      (*tL_Trigger_EventTime := UInt64Add64(ULINT_TO_ULARGE(tL_Sensor_TimeStamp), LREAL_TO_UINT64(fI_TriggerDistance/fI_ConveyorSpeed * 1E9));*)
        tL_Trigger_EventTime := (tL_Sensor_TimeStamp + LREAL_TO_ULINT(fI_TriggerDistance / fI_ConveyorSpeed * 1E9));
        iL_StartPos          := iI_CurrentPos;
      END_IF;

      cO_Activate     := cL_INACTIVE;
    END_IF;

    bO_Trigger        := TRUE;
    bO_Active         := TRUE;
  	bL_InhibitTrigger := TRUE;

  cL_WAITALMOSTSTART: (*Only active when bI_UsePositionTrigger=TRUE: wait until Start position almost reached, then set timestamp*)
    (*Remaining distance in [m], converted to REAL to avoid integer wrap problems*)
    fL_RemDist             := fI_TriggerDistance + (DINT_TO_REAL(iL_StartPos) - DINT_TO_REAL(iI_CurrentPos))*0.0254 / INT_TO_REAL(iI_Resolution);
    fL_PreTriggerPosition  := fC_PreTrigFactor * fL_DeltaTimeStamp * fI_ConveyorSpeed;

    IF fL_RemDist < fL_PreTriggerPosition THEN
      cL_State             := cL_WAITSTART;
    (*tL_Trigger_EventTime := UInt64Add64(ULINT_TO_ULARGE(tL_Sensor_TimeStamp), LREAL_TO_UINT64(fL_RemDist/fI_ConveyorSpeed * 1E9));*)
      tL_Trigger_EventTime := (tL_Sensor_TimeStamp + LREAL_TO_ULINT(fL_RemDist / fI_ConveyorSpeed * 1E9));
      cO_Activate          := cL_ACTIVE;  (*Arm EL2252*)
    ELSE
      cL_State     := cL_WAITALMOSTSTART;
      cO_Activate  := cL_INACTIVE;
    END_IF;
    bO_Trigger     := TRUE;
    bO_Active      := TRUE;

  cL_WAITSTART:       (*Wait until start time reached*)
  (*IF (UInt64Cmp64(tL_Trigger_EventTime, ULINT_TO_ULARGE(tL_CurrentTime)) = -1) THEN (* StartTime elapsed *)*)
    IF (tL_Trigger_EventTime < tL_CurrentTime) THEN (* StartTime elapsed *)
      cL_State     := cL_TRIGACTIVE;
      cO_Activate  := cL_INACTIVE; (*Disarm EL2252, trigger generated*)
    ELSE
      cL_State     := cL_WAITSTART;
      cO_Activate  := cL_ACTIVE;   (*Arm EL2252*)
    END_IF;

    bO_Trigger     := TRUE;
    bO_Active      := TRUE;

  cL_TRIGACTIVE:   (*Trigger high*)
    cL_State       := cL_WAITSTOP;

  (*tL_Trigger_EventTime := UInt64Add64(tL_Trigger_EventTime,LREAL_TO_UINT64(fL_TriggerLength*1E9));*)
    tL_Trigger_EventTime := (tL_Trigger_EventTime + LREAL_TO_ULINT(fL_TriggerLength * 1E9));

    cO_Activate    := cL_INACTIVE;
    bO_Trigger     := FALSE;
    bO_Active      := TRUE;

  cL_WAITSTOP:  (*Wait until trigger time has elapsed*)
  (*IF (UInt64Cmp64(tL_Trigger_EventTime, ULINT_TO_ULARGE(tL_CurrentTime)) = -1) THEN (* StopTime elapsed *)*)
    IF (tL_Trigger_EventTime < tL_CurrentTime) THEN (* StopTime elapsed *)
      cL_State     := cL_IDLE;
      cO_Activate  := cL_INACTIVE; (*Disarm EL2252, trigger generated*)
    ELSE
      cL_State     := cL_WAITSTOP;
      cO_Activate  := cL_ACTIVE;   (*Arm EL2252*)
    END_IF;

    bO_Trigger     := FALSE;
    bO_Active      := TRUE;

  ELSE  (*Default*)
    cL_State       := cL_IDLE;
    bO_Trigger     := FALSE;
    bO_Active      := FALSE;
    cO_Activate    := cL_INACTIVE;
END_CASE;

tO_Trigger_StartTime := tL_Trigger_EventTime;

(*Release inhibit trigger*)
bL_ReleaseInhibitTrigger := (iI_CurrentPos >= (iL_StartPos + iL_SubstrateLength));
fb_FTrig_ManualTeach(CLK := bI_ManualTeachTrigger);

IF ( bL_ReleaseInhibitTrigger OR fb_FTrig_ManualTeach.Q)
   AND bL_InhibitTrigger
THEN
	bL_InhibitTrigger := FALSE;
END_IF;

(********************************* END OF FB *****************************************************)

END_FUNCTION_BLOCK

// ---- POUs/Print/DefGrid/FB_ContainerDefGrid.TcPOU
FUNCTION_BLOCK FB_ContainerDefGrid EXTENDS FB_ContainerBase
VAR_INPUT
END_VAR
VAR_OUTPUT
END_VAR
VAR
  fBImageDeformation : FB_ImageDeformation;
END_VAR

fBImageDeformation();                       // call run cyclic image deformation

METHOD AbortDeformation : BOOL
VAR_INPUT
  sReason   : STRING;
  Src       : REFERENCE TO T_ErrSrc;
  bHideLog  : BOOL;
END_VAR
IF NOT bHideLog THEN
  LogWarning(F_Concat4('Abort deformation: ', sReason, ' Src: ', Src.aDescr));  // log reason
END_IF
setError(ErrDef:=EC_DefGrid.ecDefGrid_DefGridAbort, Src:=Src); // tag ct as error
fBImageDeformation.abort();  // abort deformation
StopScript(iCT:=THIS^);
END_METHOD

METHOD AddCamPoint : BOOL
VAR_INPUT
  sPoint : ST_DeformationPointAccurate;
END_VAR
AddCamPoint := fBImageDeformation.addCamPoint(sNewPoint:=sPoint);
END_METHOD

PROPERTY bLimited : BOOL
GET
bLimited := fBImageDeformation.bDeformationGridLimited;
END_GET
SET
fBImageDeformation.bDeformationGridLimited := bLimited;
END_SET
END_PROPERTY

(*
  Create a container, build very basics.
*)
METHOD Create : BOOL
VAR_INPUT
	nCTId	            : DINT;     (* a container identifier *)
	nCTIndex	        : UDINT;	  (* memory index (array index if CT in CT array) *)
END_VAR
SUPER^.Create(nCTId:=nCTId, nCTIndex:=nCTIndex);
fBImageDeformation.reset();
fBImageDeformation.nProcessId := THIS^.pCT^.iId;
END_METHOD

PROPERTY eCamMode : E_CameraMode
GET
eCamMode := fBImageDeformation.eCamMode;
END_GET
END_PROPERTY

(*
  Shift in x [SubPx]
*)
PROPERTY fDxShift : LREAL
GET
VAR
  errCtr : UDINT;
END_VAR
fDxShift := fBImageDeformation._nDxShift;
END_GET
END_PROPERTY

(*
  Shift in y [Px]
*)
PROPERTY fDyShift : LREAL
GET
VAR
  errCtr : UDINT;
END_VAR
fDyShift := fBImageDeformation._nDyShift;
END_GET
END_PROPERTY

PROPERTY fPrintLengthEffective : LREAL
GET
fPrintLengthEffective := fBImageDeformation.fPrintLengthEffective;
END_GET
SET
fBImageDeformation.fPrintLengthEffective := fPrintLengthEffective;
END_SET
END_PROPERTY

(*
  get a deformation point.
  :returns: TRUE if successful
*)
METHOD getDeformationPoint : BOOL;
VAR_INPUT
  nCol : UDINT;   // col select
  nRow : UDINT;   // row select
  nSel : UDINT;   // table selection
END_VAR
VAR_OUTPUT
  sPoint : ST_DeformationPointAccurate;
  bWasSet : BOOL;           // point was set by deformation
END_VAR
getDeformationPoint := fBImageDeformation.getDeformationPoint(nCol:=nCol, nRow:=nRow, nSel:=nSel, sPoint=>sPoint, bWasSet=>bWasSet);
END_METHOD

(*
  Deformation state of CT.
  :return:  TRUE in case of error -> any deformation error
*)
METHOD getDeformationStatus : BOOL
VAR_INPUT
END_VAR
VAR_OUTPUT
  eDStep: E_DeformationStep;// deformation step
  bDone : BOOL;             // deformation done
  bBusy : BOOL;             // deformation is busy
  nErrorId : UDINT;         // error id in case of error
  tExecutionTime : TIME;    // script update execution time?
  bAborted : BOOL;          // deformation is aborted/error
END_VAR
getDeformationStatus := fBImageDeformation.bError;

eDStep:= fBImageDeformation.eStep;
bBusy := fBImageDeformation.bBusy;
bDone := fBImageDeformation.bDone;
nErrorId := fBImageDeformation.nErrorId;
tExecutionTime := fBImageDeformation.tExecutionTime;
bAborted := fBImageDeformation.bAborted;
END_METHOD

PROPERTY LogLevel : E_LogSeverity
GET
LogLevel := SUPER^.LogLevel;
END_GET
SET
fBImageDeformation.LogLevel := LogLevel;
SUPER^.LogLevel := LogLevel;
END_SET
END_PROPERTY

PROPERTY nAvailableGridCols : UDINT
GET
nAvailableGridCols := fBImageDeformation._nGridCols;
END_GET
END_PROPERTY

PROPERTY nAvailableGridPoints : UDINT
GET
nAvailableGridPoints := fBImageDeformation.nAvailableGridPoints;
END_GET
END_PROPERTY

PROPERTY PUBLIC nRegisteredCameraPoints : UDINT
GET
nRegisteredCameraPoints := fBImageDeformation._nCamPoints;
END_GET
END_PROPERTY

PROPERTY pImageDeformation : POINTER TO FB_ImageDeformation
GET
pImageDeformation := ADR(fBImageDeformation);
END_GET
END_PROPERTY

PROPERTY sDefGridSettings : ST_DefGridSettings
GET
sDefGridSettings := fBImageDeformation.sDefGridSettings;
END_GET
END_PROPERTY

METHOD StartCamera
VAR_INPUT
  eCameraMode  : E_CameraMode;   // used camera mode
  fFeatureGrid : LREAL;          // deformation module update interval [Px]
  bResetDeformation : BOOL;      // reset current deformation state
END_VAR
// reset old deformation
IF bResetDeformation THEN
  fBImageDeformation.reset();
END_IF

// update mode
fBImageDeformation.eCamMode := eCameraMode;
fBImageDeformation.fFeatureGrid := fFeatureGrid;
fBImageDeformation.eStep := E_DeformationStep.cameraStarted;
END_METHOD

METHOD StartDeformation
VAR_INPUT
  sDefGridSettings : ST_DefGridSettings;
  fStartDeformationPos : LREAL;   // reference start position in [px]
END_VAR
fBImageDeformation.sDefGridSettings := sDefGridSettings;                  // apply grid setting
fBImageDeformation.startDeformation(                                      // start deformation process
  fStartDefPos:=fStartDeformationPos,     // reference position at current position [Px]
  fImageLength:=pJob^.fImageDepth / 1000        // fSubstrateDepth            //update with intended length
);
END_METHOD

METHOD StartScript
VAR_INPUT
  iDeformationHandler : I_DeformationHandler;
END_VAR
fBImageDeformation.iDeformationHandler := iDeformationHandler;
fBImageDeformation.eStep := E_DeformationStep.createdScriptContainer;
END_METHOD

METHOD StopScript : BOOL
VAR_INPUT
  iCT : I_CT;
END_VAR
IF fBImageDeformation.iDeformationHandler <> 0 THEN
  fBImageDeformation.iDeformationHandler.DeleteCachedCt(iCT:=iCT);
  fBImageDeformation.iDeformationHandler := 0; // remove handler after stopping (prevent further calls on same CT)
END_IF
END_METHOD

(*
  save a streamed deformation point.
  :returns: TRUE if successful
*)
METHOD storeStreamedDeformationPoint : BOOL;
VAR_INPUT
  pPoint : POINTER TO ST_DeformationPointAccurate;
END_VAR
IF pPoint = 0 THEN RETURN; END_IF

storeStreamedDeformationPoint := fBImageDeformation.storeStreamedDeformationPoint(pPoint:=pPoint);
END_METHOD

METHOD UpdateDeformation
VAR_INPUT
  fPos : LREAL; // relative deformation position in [px]
END_VAR
fBImageDeformation.updateDeformation(fPos:=fPos);
END_METHOD

END_FUNCTION_BLOCK

// ---- POUs/Print/DefGrid/FB_ImageDeformation.TcPOU
FUNCTION_BLOCK FB_ImageDeformation EXTENDS FB_PythonDeformation
VAR
  _eDeformationStep : E_DeformationStep;    // current active deformation step (handler)
  _eCameraMode      : E_CameraMode;         // active deformation mode
  _fFeatureGrid     : LREAL;                // camera feature grid [Px]
  _iDefHandler      : I_DeformationHandler; // deformation handler interface for global deformation control
  _nImgProcPoints   : DINT;                 // to calc gloabl dx/dy
  _nDxShift, _nDxSum : LREAL;               // global x grid shift
  _nDyShift, _nDySum : LREAL;               // global y grid shift
  
  // Cam points (stored locally)
  _nCamPoints        : UDINT;
  _sCamPoints        : ARRAY[0..100] OF ST_CameraPointTbl;   // received cam points
  _nCamPoint_MaxRefX : LREAL;               // max. x position of all available cam points [px]

  _sDefGridSettings  : ST_DefGridSettings;  // local copy of settings  
  // local DefGrid table [calculated]
  _sDefGridPoints    : ARRAY[0..nMAX_COLS_DEFGRID, 0..nMAX_ROWS_DEFGRID] OF ST_DeformationPointTbl; // [col, row] local grid point table
  _nGridPoints       : UDINT;               // stored and available grid points
  _nGridCols         : UDINT;               // count current complete grid columns
  // local DefGrid table [streamed]
  _sDefGridPointsStreamed : ARRAY[0..nMAX_COLS_DEFGRID, 0..nMAX_ROWS_DEFGRID] OF ST_DeformationPointTbl; // [col, row] local grid point table 
  _nGridRowsStreamed, _nGridColsStreamed : UDINT;
  
  // local grid handler(s) helper
  _nLocalGridColsGenerated: UDINT;          // already generated "local" grid columns XYR [0..x]

  _fStartDeformPos  : LREAL;                // position [Px] where deformation started on ct
  _nUpdatedGridCol  : UDINT;                // already updated grid column
  _nUpdatedFeature  : UDINT;                // number of updated features (a distance)
  _fPrintLengthOriginal  : LREAL;           // intended image depth in [m]
  _fPrintLengthEffective : LREAL;           // effective detected printing length in [m] (not yet used, but could be used for more accureate dx calculation in the future)
  _bDeformationGridLimited : BOOL;              // some deformation points were limited to a min/max boundary
  // others
  _nErrorId         : UDINT := 0;
  _sTempPoint       : ST_DeformationPointAccurate; 
END_VAR
VAR_STAT
  // sim
  eTestGridSelection : E_GridTypeSelection;
  nTestGridFactor : LREAL := 20;
END_VAR
VAR CONSTANT
  tPYTHON_TIMEOUT   : TIME  := T#500MS;     // python deformation script update response timeout  
  nMAX_COLS_DEFGRID : UDINT := 100;         // if you update this value you need to update the array variables as well (there we can't use this constant (beckhoff bug in table view))
  nMAX_ROWS_DEFGRID : UDINT := 100;         // if you update this value you need to update the array variables as well (there we can't use this constant (beckhoff bug in table view))
  nMAX_CAM_POINTS   : UDINT := 100;         // if you update this value you need to update the array variables as well (there we can't use this constant (beckhoff bug in table view))
END_VAR

IF NOT bInitialized THEN
  init();
END_IF

IF bUsePy THEN
  ExecPy();       // call python deformation handler
  
  // pull all GridPoints from FIFO and store to local table
  WHILE PopDeformationPoint(sNewPoint=>_sTempPoint) DO
    storeDeformationPoint(sPoint:=_sTempPoint);    // save point to table
  END_WHILE
END_IF

METHOD abort : BOOL
VAR_INPUT
END_VAR
_bAborted := TRUE;
END_METHOD

METHOD addCamPoint : BOOL
VAR_INPUT
  sNewPoint : ST_DeformationPointAccurate;
END_VAR
VAR
  sPointPx  : ST_DeformationPoint;
END_VAR
IF bUsePy THEN
  // push point to fifo for script
  
  addCamPoint := PushDeformationPoint(
                      sPoint:=F_EncodeDeformationPoint(sPoint:=sNewPoint, nResolution:=GVL_Deformation.nC_GridSubReso)
                 );
ELSE
  addCamPoint := TRUE;
END_IF

// store it to local table
IF addCamPoint THEN
  storeCameraPoint(sPoint:=sNewPoint); // store locally
END_IF
END_METHOD

PROPERTY bAborted : BOOL
GET
bAborted := _bAborted;
END_GET
END_PROPERTY

PROPERTY bBusy : BOOL
GET
bBusy := bPythonBusy AND NOT _bAborted;
END_GET
END_PROPERTY

PROPERTY bDeformationGridLimited : BOOL
GET
bDeformationGridLimited := _bDeformationGridLimited;
END_GET
SET
_bDeformationGridLimited := bDeformationGridLimited;
END_SET
END_PROPERTY

PROPERTY bDone : BOOL
GET
bDone := bPythonDeformationDone OR _bAborted OR (eStep = E_DeformationStep.nothing);
END_GET
END_PROPERTY

PROPERTY bError : BOOL
GET
bError := bPythonError OR _bAborted;
END_GET
END_PROPERTY

PROPERTY PRIVATE bUsePy : BOOL
GET
IF _sDefGridSettings.eDeformationType=E_DeformationType.ScriptGrid OR _sDefGridSettings.eDeformationType = E_DeformationType.ScriptGridTrend THEN
  bUsePy := TRUE;
END_IF
END_GET
END_PROPERTY

METHOD dumpGrid : BOOL
VAR_INPUT
END_VAR
END_METHOD

PROPERTY eCamMode : E_CameraMode
GET
eCamMode := _eCameraMode;
END_GET
SET
_eCameraMode := eCamMode;
END_SET
END_PROPERTY

PROPERTY eStep : E_DeformationStep
GET
eStep := _eDeformationStep;
END_GET
SET
IF eStep > _eDeformationStep THEN
  LogLvl(Lvl:=E_LogSeverity.Detail, Msg:=F_Concat4('Change deformation step: ', TO_STRING(_eDeformationStep), '->', TO_STRING(eStep)));
  _eDeformationStep := eStep;
END_IF
END_SET
END_PROPERTY

(*
  Camera feature grid. Section distance where points are detected and sent as group to PLC.
*)
PROPERTY fFeatureGrid : LREAL
GET
fFeatureGrid := _fFeatureGrid;
END_GET
SET
_fFeatureGrid := fFeatureGrid;
END_SET
END_PROPERTY

PROPERTY fPrintLengthEffective : LREAL
GET
fPrintLengthEffective := _fPrintLengthEffective;
END_GET
SET
_fPrintLengthEffective := fPrintLengthEffective;
END_SET
END_PROPERTY

// get neighbour camera point
// :returns: TRUE if present
METHOD PRIVATE getCamNeighbourPoint : BOOL
VAR_INPUT
  fPos    : LREAL;   // [px]
  nOffset : DINT;    // 0=previous, 1=next
END_VAR
VAR_OUTPUT
  Pn : ST_CameraPointTbl;
END_VAR
VAR
  i : DINT;
  foundIdx : DINT;
END_VAR
foundIdx := -1;
FOR i:=0 TO TO_DINT(_nCamPoints)-1 DO
  // previous search
  IF nOffset = 0 THEN
    IF _sCamPoints[i].sPoint.x_ref <= fpos THEN
      foundIdx := i;
    ELSE
      EXIT;
    END_IF
    
  // next searchs  
  ELSIF nOffset = 1 THEN
    IF _sCamPoints[i].sPoint.x_ref > fpos THEN
      foundIdx := i;
      EXIT;
    END_IF
  END_IF
END_FOR

IF foundIdx >= 0 THEN
  Pn := _sCamPoints[foundIdx];
  getCamNeighbourPoint := TRUE;  
END_IF
END_METHOD

// get neighbour camera point
// :returns: TRUE if present
METHOD getCamPointX : BOOL
VAR_INPUT
  nIdx : UDINT;    // 0=last, 1=first, 2=second
END_VAR
VAR_OUTPUT
  Pn : ST_CameraPointTbl;
END_VAR
IF nIdx = 0 THEN
  Pn := _sCamPoints[_nCamPoints-1];  // return first cam point
  getCamPointX := TRUE;
ELSIF nIdx <= _nCamPoints THEN
  Pn := _sCamPoints[nIdx-1];
  getCamPointX := TRUE;
ELSE
  //error
  Pn := _sCamPoints[0];   // error return first as fallback 
END_IF
END_METHOD

(*
  get a deformation point.
  :returns: TRUE if successful
*)
METHOD getDeformationPoint :  BOOL;
VAR_INPUT
  nCol : UDINT;   // col select
  nRow : UDINT;   // row select
  nSel : UDINT;   // table selection 0=GeneratedGrid, 1=StreamedGrid
END_VAR
VAR_OUTPUT
  sPoint : ST_DeformationPointAccurate;
  bWasSet : BOOL;
END_VAR
getDeformationPoint := FALSE;

IF TO_UDINT(nCol) > nMAX_COLS_DEFGRID THEN LogError(F_Concat5('getDeformationPoint: point col=', TO_STRING(nCol), ' out of table > ', TO_STRING(nMAX_COLS_DEFGRID), '')); RETURN; END_IF
IF TO_UDINT(nRow) > nMAX_ROWS_DEFGRID THEN LogError(F_Concat5('getDeformationPoint: point row=', TO_STRING(nRow), ' out of table > ', TO_STRING(nMAX_ROWS_DEFGRID), '')); RETURN; END_IF

IF nSel = 1 THEN
  sPoint  := _sDefGridPointsStreamed[nCol, nRow].sPoint;
  bWasSet := _sDefGridPointsStreamed[nCol, nRow].bSet;  
ELSE
  sPoint  := _sDefGridPoints[nCol, nRow].sPoint;
  bWasSet := _sDefGridPoints[nCol, nRow].bSet;  
END_IF

getDeformationPoint := TRUE;
END_METHOD

METHOD PROTECTED gridImgProc
VAR_INPUT
  pNewDeformationPoint	: POINTER TO ST_DeformationPointAccurate;
END_VAR
IF pNewDeformationPoint = 0 THEN RETURN; END_IF

_nDxSum := (_nDxSum + pNewDeformationPoint^.dx);
_nDySum := (_nDySum + pNewDeformationPoint^.dy);
IF _nImgProcPoints > 0 THEN
  _nDxShift := _nDxSum / _nImgProcPoints;
  _nDyShift := _nDySum / _nImgProcPoints;
END_IF
_nImgProcPoints := _nImgProcPoints + 1;
END_METHOD

PROPERTY iDeformationHandler : I_DeformationHandler
GET
iDeformationHandler := _iDefHandler;
END_GET
SET
_iDefHandler := iDeformationHandler;
END_SET
END_PROPERTY

METHOD init
VAR_INPUT
END_VAR
_fbTimeout.PT := tPYTHON_TIMEOUT;
bInitialized := TRUE;
END_METHOD

PROPERTY nAvailableCamPoints : UDINT
GET
nAvailableCamPoints := _nCamPoints;
END_GET
END_PROPERTY

PROPERTY nAvailableGridPoints : UDINT
GET
nAvailableGridPoints := _nGridPoints;
END_GET
END_PROPERTY

PROPERTY nErrorId : UDINT
GET
nErrorId := _nErrorId;
END_GET
END_PROPERTY

PROPERTY nProcessId : DINT
GET
nProcessId := nPythonId;
END_GET
SET
nPythonId := nProcessId;
END_SET
END_PROPERTY

METHOD reset
VAR_INPUT
END_VAR
SUPER^.Reset();   // reset FB_PythonDeformation

_nGridPoints := 0;
_nGridCols := 0;
_nCamPoints := 0;
_nCamPoint_MaxRefX := 0;
MEMSET(destAddr:=ADR(_sDefGridPoints), fillByte:=0, n:=SIZEOF(_sDefGridPoints));
MEMSET(destAddr:=ADR(_sCamPoints), fillByte:=0, n:=SIZEOF(_sCamPoints));
MEMSET(destAddr:=ADR(_sDefGridSettings), fillByte:=0, n:=SIZEOF(_sDefGridSettings));

MEMSET(destAddr:=ADR(_sDefGridPointsStreamed), fillByte:=0, n:=SIZEOF(_sDefGridPointsStreamed));
_nGridRowsStreamed := 0;
_nGridColsStreamed := 0;

_eDeformationStep := E_DeformationStep.nothing;
_eCameraMode := E_CameraMode.NoCorrection;
_iDefHandler := 0;
_nImgProcPoints   := 0;
_nDxShift         := 0;
_nDyShift         := 0;
_nDxSum           := 0;
_nDySum           := 0; 

_nLocalGridColsGenerated:=0;
_fStartDeformPos:=0;
_nUpdatedGridCol := 0;
_nUpdatedFeature := 0;
_nErrorId := 0;
_tExecutionTime := T#0s;
END_METHOD

PROPERTY sDefGridSettings : ST_DefGridSettings
GET
sDefGridSettings := _sDefGridSettings;
END_GET
SET
_sDefGridSettings := sDefGridSettings;
END_SET
END_PROPERTY

METHOD startDeformation
VAR_INPUT
  fStartDefPos : LREAL;  // [Px]
  fImageLength : LREAL;  // [m] original image length
END_VAR
_fStartDeformPos := fStartDefPos;
_fPrintLengthOriginal := fImageLength;
_fPrintLengthEffective := fImageLength;
_nUpdatedGridCol := 0;
_nUpdatedFeature := 0;
_nCamPoint_MaxRefX := 0;

eStep := E_DeformationStep.gridStarted;  // signal to start deformation (update process)
END_METHOD

METHOD PRIVATE storeCameraPoint
VAR_INPUT
  sPoint : ST_DeformationPointAccurate;
END_VAR
// save point with checks and log.

//-- check table overflow
IF _nCamPoints >= nMAX_CAM_POINTS THEN LogError(F_Concat3('storeCamPoint: array overflow ', TO_STRING(_nCamPoints), ' ignore point, ')); RETURN; END_IF

//-- store point
_sCamPoints[_nCamPoints].bSet := TRUE;
_sCamPoints[_nCamPoints].sPoint := sPoint;
_sCamPoints[_nCamPoints].tTime := F_GetCurDcTaskTime64();
_nCamPoints := _nCamPoints+1;

// -- max. x pos 
IF sPoint.x_ref > _nCamPoint_MaxRefX THEN
  _nCamPoint_MaxRefX := sPoint.x_ref;  // point most far in ct
END_IF
END_METHOD

METHOD PRIVATE storeDeformationPoint
VAR_INPUT
  sPoint : ST_DeformationPointAccurate;
END_VAR
// do global point img processing
gridImgProc(pNewDeformationPoint:=ADR(sPoint));

// save point with checks and log.
//-- check table overflow
IF TO_UDINT(sPoint.col) > nMAX_COLS_DEFGRID THEN LogError(F_Concat5('point col=', TO_STRING(sPoint.col), ' exceeds max=', TO_STRING(nMAX_COLS_DEFGRID), ' ignore point')); RETURN; END_IF
IF TO_UDINT(sPoint.row) > nMAX_ROWS_DEFGRID THEN LogError(F_Concat5('point row=', TO_STRING(sPoint.row), ' exceeds max=', TO_STRING(nMAX_ROWS_DEFGRID), ' ignore point')); RETURN; END_IF
  
//-- store point
_sDefGridPoints[sPoint.col, sPoint.row].bSet := TRUE;
_sDefGridPoints[sPoint.col, sPoint.row].sPoint := sPoint;
_sDefGridPoints[sPoint.col, sPoint.row].tTime := F_GetCurDcTaskTime64();
IF sPoint.x_ref = 0 THEN _sDefGridPoints[sPoint.col, sPoint.row].sPoint.x_ref := sPoint.col * TO_DINT(_sDefGridSettings.nGridPitchX); END_IF// calc x pos of grid point (if not done by script)
IF sPoint.y_ref = 0 THEN _sDefGridPoints[sPoint.col, sPoint.row].sPoint.y_ref := sPoint.row * TO_DINT(_sDefGridSettings.nGridPitchY); END_IF// calc x pos of grid point (if not done by script)
// count grid points 
_nGridPoints := _nGridPoints + 1;
// count current complete grid columns
IF _sDefGridSettings.nGridSizeY > 0 THEN
  _nGridCols := (_nGridPoints/_sDefGridSettings.nGridSizeY);
END_IF
END_METHOD

METHOD storeStreamedDeformationPoint : BOOL
VAR_INPUT
  pPoint : POINTER TO ST_DeformationPointAccurate;
END_VAR
IF pPoint = 0 THEN RETURN; END_IF
IF TO_UDINT(pPoint^.col) > nMAX_COLS_DEFGRID THEN RETURN; END_IF
IF TO_UDINT(pPoint^.row) > nMAX_ROWS_DEFGRID THEN RETURN; END_IF

_sDefGridPointsStreamed[pPoint^.col, pPoint^.row].bSet := TRUE;
_sDefGridPointsStreamed[pPoint^.col, pPoint^.row].sPoint := pPoint^;
_sDefGridPointsStreamed[pPoint^.col, pPoint^.row].tTime := F_GetCurDcTaskTime64();
IF pPoint^.x_ref = 0 THEN _sDefGridPointsStreamed[pPoint^.col, pPoint^.row].sPoint.x_ref := pPoint^.col * TO_DINT(_sDefGridSettings.nGridPitchX); END_IF// calc x pos of grid point (if not done by script)
IF pPoint^.y_ref = 0 THEN _sDefGridPointsStreamed[pPoint^.col, pPoint^.row].sPoint.y_ref := pPoint^.row * TO_DINT(_sDefGridSettings.nGridPitchY); END_IF// calc x pos of grid point (if not done by script)
_nGridColsStreamed := MAX(_nGridColsStreamed, TO_UDINT(pPoint^.col));
_nGridRowsStreamed := MAX(_nGridRowsStreamed, TO_UDINT(pPoint^.row));

storeStreamedDeformationPoint := TRUE;
END_METHOD

PROPERTY tExecutionTime : TIME
GET
tExecutionTime := _tExecutionTime;  // TODO: in case of local processor read other execution time
END_GET
END_PROPERTY

METHOD updateDeformation
VAR_INPUT
  fPos : LREAL;  // current CT position in [px]
END_VAR
VAR
  fPosRel_Deform      : LREAL;    // position relative to start deformation [px]
  fPosRel_CamFeature  : LREAL;    // theoretical feature position [feature nr](based on StartDeformation NOT real on camera)
  fPosRel_GridCol     : LREAL;    // current deformation grid number [grid nr]
  sPoint : ST_DeformationPoint;
  nCurrentCol, nCurrentFeature : UDINT;
END_VAR
// cyclic call and update deformation script
// - parameter checks
IF eStep < E_DeformationStep.gridStarted OR bDone THEN RETURN; END_IF  // nothing to do if deformation was not started
IF _sDefGridSettings.nGridSizeX = 0 THEN RETURN; END_IF
IF fFeatureGrid = 0 THEN fFeatureGrid := 1024; END_IF         // set some valid default (prevents division crash)

// - calc relative Deformation position
fPosRel_Deform     := fPos - _fStartDeformPos;
fPosRel_CamFeature := fPosRel_Deform / _fFeatureGrid;
fPosRel_GridCol    := fPosRel_Deform / _sDefGridSettings.nGridPitchX;

// - check available cam points --> current feature
//    Is this blocking when position is retracting?
IF FLOOR(fPosRel_CamFeature) > _nUpdatedFeature   // by CameraFeature pitch (to sync with reception of cam points)
   //FLOOR(fPosRel_GridCol) > _nUpdatedGridCol    // by Grid Pitch  // AND _nUpdatedGridCol <= _sDefGridSettings.nGridSizeX
THEN

  nCurrentCol := TO_UDINT(FLOOR(fPosRel_GridCol));
  nCurrentFeature :=  TO_UDINT(FLOOR(fPosRel_CamFeature));

  // debug info
  LogLvl(Lvl:=E_LogSeverity.Debug, Msg:=
    F_Concat6(
        F_Concat2('update at: ', TO_STRING(fPosRel_Deform)),
        F_Concat3(' feature(', TO_STRING(fPosRel_CamFeature), ')'),
        F_Concat2(' CamP: ', TO_STRING(_nCamPoints)),
        F_Concat2(' maxX: ', TO_STRING(_nCamPoint_MaxRefX)),
        F_Concat2(' GridP: ', TO_STRING(_nGridPoints)),
        F_Concat2(' at Col: ', TO_STRING(nCurrentCol))
    )
  );

  // - update Grid (py or local) with desired position
  IF bUsePy THEN
    IF _nCamPoints > 2 THEN
      UpdatePy(fPosition:=fPosRel_Deform);
      _nUpdatedGridCol := nCurrentCol;
      _nUpdatedFeature := nCurrentFeature;
    END_IF
  ELSIF _sDefGridSettings.eDeformationType = E_DeformationType.LocalMarks1D THEN
    updateLocal_1D_Marks(nGridCol:=nCurrentCol, nFeatureCt:=nCurrentFeature);
    _nUpdatedGridCol := nCurrentCol;
    _nUpdatedFeature := nCurrentFeature;
  END_IF
END_IF
END_METHOD

METHOD PRIVATE updateLocal_1D_Marks : BOOL
VAR_INPUT
  nGridCol : UDINT;
  nFeatureCt : UDINT;
END_VAR
VAR
  row, col : UDINT;
  ct : DINT;
  col_pos_px : LREAL;   // column position in [px]
  sTmpPoint : ST_DeformationPointAccurate;
  dx, dy : LREAL;
  generateGridForCol : BOOL;
  Pn0, Pn1 : ST_CameraPointTbl;
  pPx : POINTER TO ST_CameraPointTbl;
  bn0, bn1 : BOOL;
  bFirstCol, bLastCol : BOOL;
  fPointDist : LREAL;
  relativePosX : LREAL;
END_VAR
VAR_INST
  fTrig_Done : F_TRIG;
END_VAR
VAR CONSTANT
  fC_SignConversion : LREAL := -1; 
END_VAR
bFirstCol := SEL(nGridCol=0, FALSE, TRUE);
bLastCol  := SEL(nGridCol=_sDefGridSettings.nGridSizeX-1, FALSE, TRUE);

ct := 0;
FOR col:=_nLocalGridColsGenerated TO nGridCol DO      // loop over not yet gnerated columns 
  LogLvl(Lvl:=E_LogSeverity.Debug, Msg:= F_Concat2(F_Concat2('check grid for col: ', TO_STRING(col)), ''));
  
  col_pos_px := col * _sDefGridSettings.nGridPitchX;
  dx:=0; dy:=0;
  
  bn0 := getCamNeighbourPoint(fPos:=col_pos_px, nOffset:=0, Pn=>Pn0);
  bn1 := getCamNeighbourPoint(fPos:=col_pos_px, nOffset:=1, Pn=>Pn1);
  
  IF bn0 AND bn1 THEN
    // we have neighbour points --> interpolate displacement inbetween
    // dx/dy interpolation between previous and next cam point
    fPointDist := Pn1.sPoint.x_ref-Pn0.sPoint.x_ref;
    fPointDist := SEL(fPointDist=0, fPointDist, 1);    // avoid 0 division crash
    relativePosX := (col_pos_px-Pn0.sPoint.x_ref) / (fPointDist);    // relative position of col between two cam points
    dx := fC_SignConversion * (Pn0.sPoint.dx + (Pn1.sPoint.dx - Pn0.sPoint.dx) * relativePosX);
    dy := fC_SignConversion * (Pn0.sPoint.dy + (Pn1.sPoint.dy - Pn0.sPoint.dy) * relativePosX);
    generateGridForCol:=TRUE;
    
  ELSIF bFirstCol THEN
    // generate first col when we have a cam point -> deformation from first point
    IF    bn0 THEN dx:=fC_SignConversion*Pn0.sPoint.dx; dy:=fC_SignConversion*Pn0.sPoint.dy; generateGridForCol:=TRUE;
    ELSIF bn1 THEN dx:=fC_SignConversion*Pn1.sPoint.dx; dy:=fC_SignConversion*Pn1.sPoint.dy; generateGridForCol:=TRUE;
    END_IF
    
  ELSE
    // not framed by two points toward the end, purge colums if no valid cam point is given next
    IF nGridCol - _nLocalGridColsGenerated >= 3 OR bLastCol THEN 
      IF _nCamPoints > 1 THEN
        // calc deformation based on first and last point
        bn0 := getCamPointX(nIdx:=1, Pn=>Pn0);  // first
        bn0 := getCamPointX(nIdx:=0, Pn=>Pn1);  // last
        fPointDist := Pn1.sPoint.x_ref-Pn0.sPoint.x_ref;      // distance of the two points
        fPointDist := SEL(fPointDist=0, fPointDist, 1);                // avoid 0 division crash
        relativePosX := (col_pos_px-Pn0.sPoint.x_ref) / (fPointDist);    // relative position of col between two cam points
        dx := fC_SignConversion * (Pn0.sPoint.dx + (Pn1.sPoint.dx - Pn0.sPoint.dx) * relativePosX);
        dy := fC_SignConversion * (Pn0.sPoint.dy + (Pn1.sPoint.dy - Pn0.sPoint.dy) * relativePosX);
      ELSE
        // repeat first correction (we do not have more information)
        pPx := SEL(bn1, ADR(Pn0), ADR(Pn1));
        dx := fC_SignConversion * pPx^.sPoint.dx;
        dy := fC_SignConversion * pPx^.sPoint.dy;
      END_IF
      
      generateGridForCol := TRUE;
    END_IF    
  END_IF
  
  // SIMULATION: some test grid (overwrite calculation)
  IF eTestGridSelection <> E_GridTypeSelection.Default THEN
    CASE eTestGridSelection OF
      0: dx := dx; dy := dy;                                        // default usekeep calculated
      1: dx := dy := 0;                                             // no deformation on ct 
      2: dx := nTestGridFactor; dy := 0;                            // dx static (Factor)
      3: dx := 0; dy := nTestGridFactor;                            // dy static (Factor)
      4: dx := 0; dy := TO_LREAL(col) * nTestGridFactor;            // dx = factor * col
      5: dx := TO_LREAL(col) * nTestGridFactor; dy := 0;            // dy = factor * col
      6: dx := SEL(row=1, 0, nTestGridFactor ); dy := 0;            // dx row 1 = factor ( test BOF)
    END_CASE
    generateGridForCol := TRUE;
  END_IF  
  
  // generate grid for column  
  IF generateGridForCol THEN
    LogLvl(Lvl:=E_LogSeverity.Debug, Msg:= F_Concat6('generate grid for col: ', TO_STRING(col), ' dx=', TO_STRING(dx), '/dy=', TO_STRING(dy)));

    // check for cam points and generate grid
    FOR row:=0 TO _sDefGridSettings.nGridSizeY -1 DO    // all points per col
      //LogLvl(Lvl:=E_LogSeverity.Debug, Msg:= F_Concat2(F_Concat2('gen grid point c:', TO_STRING(col)), F_Concat2('/r:', TO_STRING(row))));
      
      // - calculate x/y shift and rotation based on available CamPoints
      sTmpPoint.index := TO_DINT(col * _sDefGridSettings.nGridSizeY + row);
      sTmpPoint.x_ref := col * _sDefGridSettings.nGridPitchX;
      sTmpPoint.y_ref := row * _sDefGridSettings.nGridPitchY;
      sTmpPoint.dx    := dx;
      sTmpPoint.dy    := dy;
      sTmpPoint.col   := TO_DINT(col);
      sTmpPoint.row   := TO_DINT(row);
      sTmpPoint.valid := TRUE;
      storeDeformationPoint(sPoint:=sTmpPoint);    // save point to table
    END_FOR
    
    _nLocalGridColsGenerated := _nLocalGridColsGenerated + 1;
  END_IF
  
END_FOR


// set state variables which would be updated in PyUpdate/PyExed
_tExecutionTime := T#2MS;
_nErrorId := 0;
bPythonError := FALSE;
bPythonBusy := SEL(_nGridPoints >= _sDefGridSettings.nGridPoints, TRUE, FALSE); // all points generated
//bPythonBusy := SEL(_nGridCols   >= _sDefGridSettings.nGridSizeX,  TRUE, FALSE);  // all columns generated

fTrig_Done(CLK:=bPythonBusy);
IF fTrig_Done.Q THEN
  ;
END_IF

bPythonDeformationDone := NOT bPythonBusy;
END_METHOD

END_FUNCTION_BLOCK

// ---- POUs/Print/DefGrid/FB_PythonDeformation.TcPOU
FUNCTION_BLOCK FB_PythonDeformation EXTENDS FB_BasePrint
VAR
  // The variables below are accessed by the Python script. Do not change their names!
  // ------------------------------------------
  //FIFO Buffers
  fbFifoCamPoints : FB_DeformationPointFIFO; // Input FIFO, do not use Pop()
	fbFifoGridPoints : FB_DeformationPointFIFO; // Output FIFO, do not use Push()

	//Handshake variables
	fPythonPosition : LREAL := 0.0; (* Current position to process - should be kept constant while Python script is executing *)
	nPythonId : DINT := 0;   (* ct id for unique trace of ct in script *)
  
	bPythonStartUpdate : BOOL := FALSE; (* Tell the script to start its execution *)
	bPythonAbort : BOOL := FALSE; (* Abort any pending operation - NOT IMPLEMENTED *)
  
	bPythonBusy : BOOL := FALSE;
	bPythonUpdateDone : BOOL := FALSE; (* Set by the script when it's done or if error occurs *)
	bPythonError : BOOL := FALSE; (* Set by the script if any error occures during execution, cleared with abort - NOT IMPLEMENTED*)
  nPythonStatus : UDINT := 0; (*Set by the script status of deformation - NOT IMPLEMENTED*)
	bPythonDeformationDone : BOOL := FALSE; (* Set by the script when deformation if finished *)
  // ------------------------------------------
  
  // internal control
  _fbTimeout : TON; (* Counter with timeout *)
	_tExecutionTime : TIME := T#0S;   (*exection time local for scoping*)
  _bAborted : BOOL;
  
END_VAR

METHOD ExecPy : BOOL
VAR_OUTPUT
  bBusy : BOOL;
  nErrId : UDINT;
END_VAR
VAR
  _sTempPoint : ST_DeformationPoint;
END_VAR
// update FIFOs (external ADS access)
fbFifoCamPoints();
fbFifoGridPoints();

// work with script
IF bPythonBusy THEN // Pending job
	IF _fbTimeout.Q THEN // Timeout occurs
		_tExecutionTime := _fbTimeout.ET;
    bPythonAbort := TRUE;   // abort (pending operation) because id did not repond within timeout
		bPythonError := TRUE;   // set internal error
		nErrId := 1;
		bPythonBusy := FALSE;
    LogError(F_Concat4('Timeout during bPythonBusy, ExecTime:', TO_STRING(_tExecutionTime), ' Err:', TO_STRING(nErrId)));
	ELSIF bPythonUpdateDone THEN //Script done
		_tExecutionTime := _fbTimeout.ET;
		bPythonBusy := FALSE;
		IF bPythonError THEN
			nErrId := 2;
      LogError(F_Concat4('Error/abort requested by py, ExecTime:', TO_STRING(_tExecutionTime), ' Err:', TO_STRING(nErrId)));
		END_IF
  ELSIF _bAborted THEN      // abort if abort request set on ct
    bPythonBusy := FALSE;
    bPythonError := TRUE;   // set internal error
    nErrId := 3;
	END_IF
ELSIF bPythonAbort THEN
	bPythonStartUpdate := FALSE;
ELSE // Update/Job done  
  bPythonAbort := FALSE;
	bPythonStartUpdate := FALSE;
	bPythonUpdateDone := FALSE;
END_IF

_fbTimeout(IN := bPythonBusy);
END_METHOD

METHOD PROTECTED PopDeformationPoint :  BOOL;
VAR_OUTPUT
  sNewPoint : ST_DeformationPointAccurate;
END_VAR
VAR
  sPoint : ST_DeformationPoint;
END_VAR
IF fbFifoGridPoints.nCount > 0 THEN
  PopDeformationPoint := fbFifoGridPoints.Pop(sGridPoint=>sPoint);
  sNewPoint := F_DecodeDeformationPoint(sPoint:=sPoint, nResolution:=GVL_Deformation.nC_GridSubReso);
ELSE
  PopDeformationPoint := FALSE;
END_IF
END_METHOD

METHOD PROTECTED PushDeformationPoint : BOOL
VAR_INPUT
  sPoint : ST_DeformationPoint;
END_VAR
PushDeformationPoint:= fbFifoCamPoints.Push(sPoint);
END_METHOD

METHOD Reset
VAR_INPUT
END_VAR
fPythonPosition := 0.0;
//nPythonId := ;
bPythonStartUpdate := FALSE;
bPythonAbort := FALSE;
bPythonBusy := FALSE;
bPythonUpdateDone := FALSE;
bPythonError := FALSE;
nPythonStatus := 0;
bPythonDeformationDone := FALSE;

_fbTimeout(IN:=FALSE);
_bAborted := FALSE;

fbFifoCamPoints.Reset();
fbFifoGridPoints.Reset();
END_METHOD

METHOD UpdatePy : BOOL
VAR_INPUT
  fPosition : LREAL;
END_VAR
IF bPythonBusy THEN // Pending job
  UpdatePy:=FALSE;
  LogLvl(Lvl:=E_LogSeverity.Debug, Msg:='Python was still busy during updateDeformation');

ELSE // Job done

  IF NOT bPythonDeformationDone AND NOT bPythonAbort THEN // Sample input
    // start a update
    fPythonPosition := fPosition * GVL_Deformation.nC_GridSubReso;
    bPythonBusy := TRUE;
    bPythonError := FALSE;

    // Start script
    bPythonStartUpdate := TRUE;      
  END_IF

  UpdatePy:=TRUE;
END_IF
END_METHOD

END_FUNCTION_BLOCK

// ---- POUs/Print/DefGrid/FB_DeformationPointFIFO.TcPOU
FUNCTION_BLOCK FB_DeformationPointFIFO
VAR_OUTPUT
	nCount    : UINT;                 // Fill level
  nBufferSize : UINT := MAX_BUFFER_SIZE;
  nBufferItemSize : UINT := BUFFER_ITEM_SIZE;
END_VAR
VAR
	sBuffer 	: ARRAY[0..(MAX_BUFFER_SIZE-1)] OF ST_DeformationPoint;
	nHeadPtr  : UINT := 0;            // Point to the first non-empty idx
	nTailPtr  : UINT := 0;            // Pointer to the first free idx
  _bError    : BOOL;
END_VAR
VAR CONSTANT
	MAX_BUFFER_SIZE   : UINT := 1000;  // max. buffer size
	BUFFER_ITEM_SIZE  : UINT := SIZEOF(ST_DeformationPoint)/4; // Divide by 4 as we packed the ST_POINT with 32bits steps
END_VAR


(* now done async in method, this was dangerous...
// FIFO level
IF nTailPtr <= nHeadPtr THEN
	nCount := nHeadPtr - nTailPtr;
ELSE
	nCount := MAX_BUFFER_SIZE + nHeadPtr - nTailPtr;
END_IF
*)

PROPERTY bError : BOOL
GET
bError := _bError;
END_GET
END_PROPERTY

(*
  Get point from fifo queue. 
  :return: TRUE on success
*)
METHOD Pop : BOOL
VAR_OUTPUT
	sGridPoint : ST_DeformationPoint;
END_VAR
IF nCount = 0 THEN
  F_LogError('FB_DeformationPointFIFO is empty, cannot return an element');
  _bError := TRUE; 
  RETURN;
END_IF

sGridPoint := sBuffer[nTailPtr];
nTailPtr := (nTailPtr + 1) MOD MAX_BUFFER_SIZE;
nCount := nCount - 1;
_bError := FALSE;
Pop := TRUE;
END_METHOD

(*
  Add a new point to the fifo queue.
  :return: TRUE on success.
*)
METHOD Push : BOOL
VAR_INPUT
	sNewPoint : ST_DeformationPoint;
END_VAR
IF nCount >= MAX_BUFFER_SIZE THEN
  F_LogError('FB_DeformationPointFIFO overflow, element ignored');
  _bError := TRUE;
  RETURN;
END_IF

sBuffer[nHeadPtr] := sNewPoint;
nHeadPtr := (nHeadPtr + 1) MOD MAX_BUFFER_SIZE;
nCount := nCount + 1;
_bError := FALSE;
Push := TRUE;
END_METHOD

METHOD Reset : BOOL
VAR_INPUT
END_VAR
nTailPtr := 0;
nHeadPtr := 0;
nCount := 0;
_bError := 0;
END_METHOD

END_FUNCTION_BLOCK

// ---- POUs/Print/DefGrid/FB_CTManagerDefGrid.TcPOU
FUNCTION_BLOCK FB_CTManagerDefGrid EXTENDS FB_CTManager
VAR
  fbContainerInstances    : ARRAY[0..nC_MAX_CTS-1] OF FB_ContainerDefGrid;   // NOTE: 0 based array like base in library
  nCtr, nIndx : UDINT;
  _LogLevelCTs : E_LogSeverity := E_LogSeverity.Info;
END_VAR

// call CT manager base
SUPER^();

// call specific CT implementation
nCtr := 0;
WHILE nCtr < nListCount DO
  nIndx := ((nListTail + nCtr) MOD nC_MAX_CTS);    // calculate element index in list
  
  // cyclic call of CT body
  fbContainerInstances[nIndx]();
  
  nCtr := nCtr + 1;
END_WHILE

updateLogLevelsCTs();

(*
  Abort CTs
*)
METHOD AbortCts : BOOL
VAR_INPUT
  iCT : I_CT;     // reference CT 
  nSel : INT;     // selection: -1=all older (created before reference), 0=current only, 1=all newer (created after reference)
  Src : REFERENCE TO T_ErrSrc;
END_VAR
VAR
  iIterCt : I_CT;
  pCtSelected : POINTER TO FB_ContainerDefGrid;
END_VAR

// WARNING: This function is NOT tested!!! 
//    TODO: remove this comments when tested

IF nSel = 0 THEN
  // Abort referenced CT
  pCtSelected := GetContainerInstance(iCT:=iCT);
  IF pCtSelected <> 0 THEN
    pCtSelected^.AbortDeformation(sReason:=F_Concat2('CTM Abort CTs Sel=', TO_STRING(nSel)), Src:=Src, bHideLog:=FALSE);
  END_IF

ELSIF nSel < 0 THEN
  // Abort previous
  iIterCt := iCT;
  WHILE iIterCt.pListPrev <> 0 DO
    // get instance and abort
    pCtSelected := GetContainerInstance(iCT:=iIterCt);
    IF pCtSelected <> 0 THEN
      pCtSelected^.AbortDeformation(sReason:=F_Concat2('CTM Abort CTs Sel=', TO_STRING(nSel)), Src:=Src, bHideLog:=FALSE);
    END_IF
    // select prev
    iIterCt := iIterCt.pListPrev;
  END_WHILE

ELSIF nSel > 0 THEN  
  // Abort next
  iIterCt := iCT;
  WHILE iIterCt.pListNext <> 0 DO
    // get instance and abort
    pCtSelected := GetContainerInstance(iCT:=iIterCt);
    IF pCtSelected <> 0 THEN
      pCtSelected^.AbortDeformation(sReason:=F_Concat2('CTM Abort CTs Sel=', TO_STRING(nSel)), Src:=Src, bHideLog:=FALSE);
    END_IF
    // select next
    iIterCt := iIterCt.pListNext;
  END_WHILE
END_IF
END_METHOD

(*
  Get specific container reference (pointer) from container interface.
*)
METHOD PUBLIC GetContainerInstance : POINTER TO FB_ContainerDefGrid
VAR_INPUT
  iCT              : I_CT;          (*container at triggered event position*)
END_VAR
VAR
  nCtSel             : UDINT;
END_VAR
IF iCT = 0 THEN LogError(Msg:='GetContainerInstance invalid container'); RETURN; END_IF
nCtSel := iCT.pCT^.nMemIndex;
IF nCtSel < nC_MAX_CTS THEN
  GetContainerInstance := ADR( fbContainerInstances[nCtSel] );
END_IF
END_METHOD

METHOD Init
VAR
  nCtr      : UDINT;
END_VAR
_LogLevelCTs := E_LogSeverity.Info;

// init FB_CTManager(base) list (interface I_CT) with specific Container instances (FBs) 
FOR nCtr := 0 TO nC_MAX_CTS-1 DO
  iContainerList[nCtr] := fbContainerInstances[nCtr];
  fbContainerInstances[nCtr].LogLevel := _LogLevelCTs;
END_FOR

// call parent init
SUPER^.InitBase(aName:='CTM', aUnit:='SubPx', bAutoDelete:=TRUE);
END_METHOD

PROPERTY sCTDefGridInstancesPath : STRING
GET
// build path tho one image deformation fb
// e.g. PRG_PRINT.fbCTM.fbContainerInstances[%id%].fBImageDeformation where %id% will be resolved later in the pyhton script.
//      array in plc lower bound is index 0
sCTDefGridInstancesPath := F_CONCAT2(THIS^.InstanceName, '.fbContainerInstances[%id%].fBImageDeformation');
END_GET
END_PROPERTY

METHOD PRIVATE updateLogLevelsCTs
VAR_INST
  _LogLvl_mem  : E_LogSeverity;
END_VAR
// logLevel update from manager to all containers
IF _LogLevelCTs <> _LogLvl_mem THEN 
  nCtr := 0;
  WHILE nCtr < nC_MAX_CTS DO
    fbContainerInstances[nCtr].LogLevel := _LogLevelCTs;
    nCtr := nCtr + 1;
  END_WHILE
END_IF

_LogLvl_mem := _LogLevelCTs;
END_METHOD

END_FUNCTION_BLOCK

// ---- POUs/Print/DefGrid/FB_CTTrackerView.TcPOU
FUNCTION_BLOCK FB_CTTrackerView
VAR_INPUT
  fX_m,  fY_m     : LREAL;            // max. x/y position [m]
  nX_px, nY_px    : DINT;             // max. x/y pixel in view
  fPxToMRatio     : LREAL;            // 
  iPrintPosition  : I_PrintPosition;  // 
END_VAR

VAR
  // helper
  bInit   : BOOL;
  nCtr    : UDINT;
  nNum    : UDINT;
  
  // config
  _pCTTracker : POINTER TO FB_CTTracker;
  _fPrintResolution : LREAL;      // [dpi]
  _fSubPixelResolution : LREAL;   // sub pixel resolution
  
  // Container view list
  iCT     : I_CT;
  aCTV    : ARRAY[1..iCPr_MAX_CONTAINER] OF FB_ContainerView;
  
  // view control
  
END_VAR
VAR CONSTANT
END_VAR

IF NOT checkConfig() THEN RETURN; END_IF    // check config

// -- show CTs -----------------------
nNum := _pCTTracker^.nCount;
FOR nCtr := 1 TO nNum DO
  // get CT interface from list
  iCT := _pCTTracker^.getCT(nIdx:=nCtr);
  IF iCT <> 0 THEN
    // set position
    aCTV[nCtr].setPos(x:=iCT.GetPosRel(iTracker:=_pCTTracker^), y:=0);

    // display
    aCTV[nCtr].bHide := FALSE;
    aCTV[nCtr]( iCT:=iCT, 
                iIdx:=UDINT_TO_UINT(iCT.pCT^.nMemIndex), 
                fPxtoMRatio:=fPxToMRatio, 
                fPosToMFactor := 0.0254 / (_fPrintResolution*_fSubPixelResolution), 
                iTracker:=_pCTTracker^);
  END_IF
END_FOR

FOR nCtr := (nNum+1) TO iCPr_MAX_CONTAINER DO
  aCTV[nCtr].iCT := 0;
  aCTV[nCtr].bHide := TRUE;
END_FOR

METHOD checkConfig : BOOL
VAR_INPUT
END_VAR
VAR_INST
  _fX_m, _fY_m   : LREAL;
  _nX_px, _nY_px : DINT; 
END_VAR
VAR
  bOK : BOOL;
END_VAR
IF NOT bInit THEN RETURN; END_IF
IF iPrintPosition = 0 THEN RETURN; END_IF

_fPrintResolution := iPrintPosition.fPrintResolution;
_fSubPixelResolution := iPrintPosition.fSubPxResolution;

// changed settings
IF _fX_m <> fX_m OR
          _fY_m <> fY_m OR
          _nX_px <> nX_px OR
          _nY_px <> nY_px THEN
  // save new config
   _fX_m := fX_m;
   _fY_m := fY_m;
   _nX_px := nX_px;
   _nY_px := nY_px;
   config();
END_IF

checkConfig := TRUE;
END_METHOD

METHOD PRIVATE config
VAR_INPUT
END_VAR
// NOTE: some config values are given only here (internally)
FOR nCtr := 1 TO iCPr_MAX_CONTAINER DO
  aCTV[nCtr].init(
    nXPosMin:=0,
    nXPosMax:= F_MeterToSubPixel(fPosMeter := fX_m, fResoSubPx := _fPrintResolution * _fSubPixelResolution),
    nYPosMin:=0,
    nYPosMax:=F_MeterToSubPixel(fPosMeter := fY_m, fResoSubPx := _fPrintResolution * _fSubPixelResolution),
    bXFlip:=TRUE,
    bYFlip:=FALSE,
    nXMinPx:=0,
    nXMaxPx:=nX_px,
    nYMinPx:=0,
    nYMaxPx:=nY_px,
  );
  aCTV[nCtr].setPos(x:=0, y:=0);
END_FOR

bInit := TRUE;
END_METHOD

METHOD init : BOOL
VAR_INPUT
  pCTTracker : POINTER TO FB_CTTracker;
END_VAR
IF pCTTracker = 0 THEN RETURN; END_IF

_pCTTracker := pCTTracker;

bInit := TRUE;
END_METHOD

END_FUNCTION_BLOCK

// ---- POUs/Print/DefGrid/FB_DropSpeedComp.TcPOU
FUNCTION_BLOCK FB_DropSpeedComp
VAR_INPUT
  fMasterSpeed         : LREAL; //[m/s]
  fDropTravelDistance  : LREAL; //[m]
END_VAR
VAR_OUTPUT
  fDropPlacementError  : LREAL;
END_VAR
VAR PERSISTENT
  _bEnable             : BOOL := TRUE;
  _fDropSpeed          : LREAL := 6;         //[m/s] DropSpeed compensation, drop speed
  _fDropSpeedDeadTime  : LREAL := 0.388889;  //[ms]  DropSpeed compensation, additional dead time
END_VAR
VAR
  bCalcDeadTime        : BOOL;
  fTestSpeed           : ARRAY[1..2] OF LREAL;  // [m/min] speed at which test was done [SpeedTest1, SpeedTest2]
  fTestDisplacement    : ARRAY[1..2] OF LREAL;  // [um] measured displacement after test [MesureTest1, MeasureTest2]
  fDiffSpeed : LREAL;
  fDiffPlace : LREAL;
END_VAR

(*Speed compensation*)
IF _bEnable AND (_fDropSpeed > 0) THEN
	fDropPlacementError :=  (  (fDropTravelDistance / _fDropSpeed)
                        + (_fDropSpeedDeadTime / 1000))             (*[s]*)
                        * fMasterSpeed;
ELSE
  fDropPlacementError := 0;
END_IF;

// calculate add/dead time
IF bCalcDeadTime THEN bCalcDeadTime := FALSE;
  calcDeadTime();
END_IF

{attribute 'monitoring':='call'}
PROPERTY bEnable : BOOL
GET
bEnable := _bEnable;
END_GET
SET
_bEnable := bEnable;
END_SET
END_PROPERTY

METHOD PRIVATE calcDeadTime : BOOL
VAR_INPUT
END_VAR
fDiffSpeed :=  ( fTestSpeed[2] - fTestSpeed[1] ) * 1/60;
fDiffPlace :=  ( fTestDisplacement[2] - fTestDisplacement[1] ) * 1/1_000_000;

IF fDiffSpeed <> 0 THEN   // avoid crash
  // calc time
  _fDropSpeedDeadTime := 
  (
      fDiffPlace      // displacement diff
    * 1/fDiffSpeed    // speed diff
  ) * 1000;           // [s] -> [ms]
ELSE
  F_LogError('DropSpeedComp invalid TestSpeed given -> DeadTime not updated');
END_IF


// reset entries
fTestSpeed[2] := fTestSpeed[1] := 0;
fTestDisplacement[2] := fTestDisplacement[1] := 0;
END_METHOD

{attribute 'monitoring':='call'}
PROPERTY fDropSpeed : LREAL
GET
fDropSpeed := _fDropSpeed;
END_GET
SET
_fDropSpeed := fDropSpeed;
END_SET
END_PROPERTY

{attribute 'monitoring':='call'}
PROPERTY fDropSpeedDeadTime : LREAL
GET
fDropSpeedDeadTime := _fDropSpeedDeadTime;
END_GET
SET
_fDropSpeedDeadTime := fDropSpeedDeadTime;
END_SET
END_PROPERTY

END_FUNCTION_BLOCK

// ---- POUs/Print/DefGrid/FB_FineAlignement.TcPOU
(*
  This fb handles mechanical print unit corrections.
  - a 4p grid distortion
  - print unit bar banana correction
  NOTE: temperature extention of whole printbar is still handled in camera
*)
FUNCTION_BLOCK FB_FineAlignement EXTENDS FB_BasePrint IMPLEMENTS I_GridPointCorrection
VAR
  // config
  _fPxResolution     : LREAL; // pixel resolution

  // corrections
  //-- 4 point PU deformation correction/distortion
  //    VISU setup point providing reference and correction (NOTE: persists settings internally)
  _fbPlcCorrPoints : ARRAY[1..4] OF FB_PointCorr;
  //-- banana correction
  _fT1 : LREAL;   // temperature 1
  _fT2 : LREAL;   // temperature 2
  _dx_middle : LREAL;  // correction in middle (for view only)
  _y_max : LREAL; // print unit width [mm]
  //-- PUC 4p correction
  _pAdsCam           : POINTER TO FB_ADS_CAMERA;  // camera interface PUC
  aPucPointNames : ARRAY[1..4] OF STRING := ['1','2','3','4'];
  
  // helper
  lCtr     : UDINT;
  
  // unit test & debug
  _bUT_4p, _bUT_banana, _bUT_4pPuc : BOOL;
  _sUTPoints_dx : ARRAY[0..nC_UT_cols, 0..nC_UT_rows] OF LREAL;
  _sUTPoints_dy : ARRAY[0..nC_UT_cols, 0..nC_UT_rows] OF LREAL;
  // 4pPUC
  bSelect : ARRAY[1..4] OF BOOL;
  bSelected : ARRAY[1..4] OF BOOL;
  nSelectedPoint : UDINT;
  bXPlus, bXMinus, bYPlus, bYMinus : BOOL;
END_VAR
VAR PERSISTENT
  //-- 4point correction
  _bEnable_4p    : BOOL := FALSE;
  _bEnablePuc_4p : BOOL := FALSE;
  //  persistence of points see: FB_PointCorr
  //-- banana correction
  _bEnable_banana : BOOL := FALSE;
  _e_max_per_deltaT : LREAL := 0.01;  // [mm/°C]  TODO: use from config
END_VAR
VAR CONSTANT
  // Unit test configuration
  nC_UT_cols : DINT := 6;   // for test only
  nC_UT_rows : DINT := 5;   // for test only
END_VAR

// cyclic caluclation and view updates
//        NOTE: deformation is happening in updateCorrection() callback

//-- 4p correction
//   visu overrides (limitation rectancular point definition)
_fbPlcCorrPoints[3].fX_Ref := _fbPlcCorrPoints[1].fX_Ref;
_fbPlcCorrPoints[4].fX_Ref := _fbPlcCorrPoints[2].fX_Ref;
_fbPlcCorrPoints[2].fY_Ref := _fbPlcCorrPoints[1].fY_Ref;
_fbPlcCorrPoints[4].fY_Ref := _fbPlcCorrPoints[3].fY_Ref;
//   update CorrectionPoints view elements
FOR lCtr := 1 TO 4 DO
  _fbPlcCorrPoints[lCtr](); 
END_FOR

//-- banana correction
// just calculate the dx in the middle of the PU, just for the VISU
calc_banana_correction(x_pos:=0, y_pos:=_y_max/(2*1000), fT1:=_fT1, fT2:=_fT2, dx_corr=>_dx_middle);
_dx_middle := _dx_middle * 1000; // [m] --> [mm] for visu

// Unit test
IF _bUT_4p THEN _bUT_4p := FALSE; _test_4p(); END_IF
IF _bUT_banana THEN _bUT_banana := FALSE; _test_banana(); END_IF
IF _bUT_4pPuc THEN _test_Puc4p(); END_IF

METHOD PRIVATE _test_4p
VAR
  sPoint : ST_DeformationPoint;
  nCol, nRow, nCrPoint : DINT;
  dx, dy : LREAL;       // correction in [m]
  dx_px, dy_px : DINT;  // correction in [px]
  pPUC_CorrPointsInd : POINTER TO ARRAY[1..4] OF ST_CORRECTION_POINT;
  
  nCorrectionX : ARRAY[1..4] OF REAL := [-0.25, -0.2, 0.35, 0.35];
  nCorrectionY : ARRAY[1..4] OF REAL := [-0.45, -0.3, -0.8, -0.65];
  nCorrectionPointX_PLC : ARRAY[1..4] OF REAL := [0, 1000,   0, 1000];
  nCorrectionPointY_PLC : ARRAY[1..4] OF REAL := [0,   0, 702, 702];
  nCorrectionPointX_PUC : ARRAY[1..4] OF REAL := [0, 671.99,   0, 671.99];
  nCorrectionPointY_PUC : ARRAY[1..4] OF REAL := [-0.0001666666, -0.0001666666, 754.2108, 754.2108];
END_VAR
// setup test correcton points location for PLC & PUC 4p testing
pPUC_CorrPointsInd := _pAdsCam^.pCorrectionPointsIndication;
IF pPUC_CorrPointsInd = 0 THEN F_Report_Error(ErrType:=EN_REPORT_ERROR_TYPE.Report_Error_0Pointer);  RETURN; END_IF

FOR nCrPoint:=1 TO 4 DO
  // correction point location
  // -- PLC
  _fbPlcCorrPoints[nCrPoint].fX_Ref := nCorrectionPointX_PLC[nCrPoint];
  _fbPlcCorrPoints[nCrPoint].fY_Ref := nCorrectionPointY_PLC[nCrPoint];
  // -- PUC  
  pPUC_CorrPointsInd^[nCrPoint].posx := nCorrectionPointX_PUC[nCrPoint];
  pPUC_CorrPointsInd^[nCrPoint].posy := nCorrectionPointY_PUC[nCrPoint];
  
  // point correction  
  // -- PLC
  _fbPlcCorrPoints[nCrPoint].fX := nCorrectionX[nCrPoint];
  _fbPlcCorrPoints[nCrPoint].fY := nCorrectionY[nCrPoint];
  // -- PUC
  pPUC_CorrPointsInd^[nCrPoint].x := nCorrectionX[nCrPoint];
  pPUC_CorrPointsInd^[nCrPoint].y := nCorrectionY[nCrPoint];
END_FOR

// generate internal test grid
FOR nCol:=0 TO nC_UT_cols DO
  FOR nRow:=0 TO nC_UT_rows DO
    sPoint.col := nCol;
    sPoint.row := nRow;
    sPoint.x_ref := nCol * TO_DINT(GVL_Deformation.nC_DefaultGridPitch_X);
    sPoint.y_ref := nRow * TO_DINT(GVL_Deformation.nC_DefaultGridPitch_Y);
    sPoint.dx := 0;   // no previous deformation
    sPoint.dy := 0;   // no previous deformation
    
    // calc 4p PLC correction and apply to point
    calc_4p_correction(
        x_pos:=F_SubPixelToMeter(lPosSubPx:=sPoint.x_ref, fResSubPx:=_fPxResolution), 
        y_pos:=F_SubPixelToMeter(lPosSubPx:=sPoint.y_ref, fResSubPx:=_fPxResolution), 
        dx_corr=>dx, 
        dy_corr=>dy);
    LogInfo(
      F_Concat4(
        '4p PLC: point:', 
        F_Concat4(' x=', TO_STRING(sPoint.x_ref), '/y=', TO_STRING(sPoint.y_ref)),
        F_Concat2(' dx=', TO_STRING(dx)),
        F_Concat2(' dy=', TO_STRING(dy))
      )
    );

    // --- store in table for verification with Excel caluculation
    dx_px := F_MeterToSubPixel(fPosMeter:=dx, fResoSubPx:=_fPxResolution);
    dy_px := F_MeterToSubPixel(fPosMeter:=dy, fResoSubPx:=_fPxResolution);
    // save corrected point
    _sUTPoints_dx[nCol, nRow] := dx_px;
    _sUTPoints_dy[nCol, nRow] := dy_px;
    // print corrected point
    LogInfo(
      F_Concat4(
        F_Concat4('[c/r] ', TO_STRING(sPoint.col), '/', TO_STRING(sPoint.row)),
        F_Concat7(' dx: ', TO_STRING(sPoint.dx), '>', TO_STRING(dx_px), ' (', TO_STRING(dx), ')'),
        F_Concat7(' dy: ', TO_STRING(sPoint.dy), '>', TO_STRING(dy_px), ' (', TO_STRING(dy), ')'),
        SEL(sPoint.dx<>dx_px OR sPoint.dy<>dy_px,'',' !!!')
      )
    );
    // ---------------------------------
    
    // calc 4p PUC correction and apply to point
    calc_PUC_4p_correction(
        x_pos:=F_SubPixelToMeter(lPosSubPx:=sPoint.x_ref, fResSubPx:=_fPxResolution), 
        y_pos:=F_SubPixelToMeter(lPosSubPx:=sPoint.y_ref, fResSubPx:=_fPxResolution), 
        dx_corr=>dx, 
        dy_corr=>dy);
    LogInfo(
      F_Concat4(
        '4p PUC: point:', 
        F_Concat4(' x=', TO_STRING(sPoint.x_ref), '/y=', TO_STRING(sPoint.y_ref)),
        F_Concat2(' dx=', TO_STRING(dx)),
        F_Concat2(' dy=', TO_STRING(dy))
      )
    );

  END_FOR  
END_FOR
END_METHOD

METHOD PRIVATE _test_banana
VAR
  sPoint : ST_DeformationPoint;
  nCol, nRow : DINT;
  dx, dy : LREAL;       // correction in [m]
  dx_px, dy_px : LREAL;  // correction in [px]
END_VAR
// generate internal grid
FOR nCol:=0 TO nC_UT_cols DO
  FOR nRow:=0 TO nC_UT_rows DO
    sPoint.col := nCol;
    sPoint.row := nRow;
    sPoint.x_ref := nCol * TO_DINT(GVL_Deformation.nC_DefaultGridPitch_X);
    sPoint.y_ref := nRow * TO_DINT(GVL_Deformation.nC_DefaultGridPitch_Y);
    sPoint.dx := 0;   // no previous deformation
    sPoint.dy := 0;   // no previous deformation
    
    // calc correction and apply to point
    calc_banana_correction(
        x_pos:=F_SubPixelToMeter(lPosSubPx:=sPoint.x_ref, fResSubPx:=_fPxResolution), 
        Y_pos:=F_SubPixelToMeter(lPosSubPx:=sPoint.y_ref, fResSubPx:=_fPxResolution),
        fT1 := 68,
        fT2 := 48, 
        dx_corr=>dx
    );
    dx_px := dx;
    dy_px := dy;
    // save corrected point (dx @y-pos)
    _sUTPoints_dx[nCol, nRow] := dx_px;
    _sUTPoints_dy[nCol, nRow] := F_SubPixelToMeter(lPosSubPx:=sPoint.y_ref, fResSubPx:=_fPxResolution)*1000;
    
    // print corrected point
    LogInfo(
      F_Concat4(
        F_Concat4('[c/r] ', TO_STRING(sPoint.col), '/', TO_STRING(sPoint.row)),
        F_Concat6(' dx: ', TO_STRING(sPoint.dx), '>', TO_STRING(TO_DINT(dx_px)), ' [', TO_STRING(dx)),
        F_Concat6('  dy: ', TO_STRING(sPoint.dy), '>', TO_STRING(TO_DINT(dy_px)), ' [', TO_STRING(dy)),
        SEL(sPoint.dx<>dx_px OR sPoint.dy<>dy_px,'',' !!!')
      )
    );
  END_FOR  
END_FOR
END_METHOD

METHOD PRIVATE _test_Puc4p
VAR
  i : UDINT;

  pPUC_CorrPointsInd : POINTER TO ARRAY[1..4] OF ST_CORRECTION_POINT;
  pPoint : POINTER TO ST_CORRECTION_POINT;
END_VAR
pPUC_CorrPointsInd := _pAdsCam^.pCorrectionPointsIndication;      // get points array from ADS
IF pPUC_CorrPointsInd = 0 THEN F_Report_Error(ErrType:=EN_REPORT_ERROR_TYPE.Report_Error_0Pointer);  RETURN; END_IF

// do selection
IF    bSelect[1] THEN bSelect[1]:=FALSE; MEMSET(destAddr:=ADR(bSelected), fillByte:=0, n:=SIZEOF(bSelected)); bSelected[1] := TRUE; nSelectedPoint:=1;
ELSIF bSelect[2] THEN bSelect[2]:=FALSE; MEMSET(destAddr:=ADR(bSelected), fillByte:=0, n:=SIZEOF(bSelected)); bSelected[2] := TRUE; nSelectedPoint:=2;
ELSIF bSelect[3] THEN bSelect[3]:=FALSE; MEMSET(destAddr:=ADR(bSelected), fillByte:=0, n:=SIZEOF(bSelected)); bSelected[3] := TRUE; nSelectedPoint:=3;
ELSIF bSelect[4] THEN bSelect[4]:=FALSE; MEMSET(destAddr:=ADR(bSelected), fillByte:=0, n:=SIZEOF(bSelected)); bSelected[4] := TRUE; nSelectedPoint:=4;
END_IF

IF    bSelected[1] THEN pPoint := ADR(pPUC_CorrPointsInd^[1]);
ELSIF bSelected[2] THEN pPoint := ADR(pPUC_CorrPointsInd^[2]);
ELSIF bSelected[3] THEN pPoint := ADR(pPUC_CorrPointsInd^[3]);
ELSIF bSelected[4] THEN pPoint := ADR(pPUC_CorrPointsInd^[4]);
ELSE                    pPoint := ADR(pPUC_CorrPointsInd^[1]);
END_IF

IF bXPlus  THEN bXPlus  := FALSE; pPoint^.x := pPoint^.x + 0.05; END_IF
IF bXMinus THEN bXMinus := FALSE; pPoint^.x := pPoint^.x - 0.05; END_IF
IF bYPlus  THEN bYPlus  := FALSE; pPoint^.y := pPoint^.y + 0.05; END_IF
IF bYMinus THEN bYMinus := FALSE; pPoint^.y := pPoint^.y - 0.05; END_IF
END_METHOD

(*
  Calculate grid point displacement for a distortion with 4 rectangular defined points.
  Uses 2-bilinear interpolation between the 4 rectancular reference points.
*)
METHOD PRIVATE calc_4p_correction : BOOL
VAR_INPUT
  x_pos   : LREAL;    // point x position [m]
  y_pos   : LREAL;    // point y position [m]
END_VAR
VAR_OUTPUT
  dx_corr : LREAL;    // point correction x [m]
  dy_corr : LREAL;    // point correction y [m]
END_VAR
VAR
  dx, dy : LREAL;     // difference between Calibration Points (rectangle)
  x1, x2, y1, y2 : LREAL;
  cx1, cx2, cy1, cy2 : LREAL;
  GPx, GPy : LREAL;
  CVx, CVy : LREAL;
  lErrCtr : UDINT;
END_VAR

// Grid point position
GPx := x_pos; 
GPy := y_pos;

// Interpolation in x
x1 := _fbPlcCorrPoints[1].fX_Ref / 1000;    // [mm -> m]
x2 := _fbPlcCorrPoints[2].fX_Ref / 1000;    // [mm -> m]
dx := x2-x1;
IF dx = 0 THEN (*F_Report_Error(ErrType:=EN_REPORT_ERROR_TYPE.Report_Error_0Pointer);*) RETURN; END_IF

cx1 := (x2-GPx)/dx * (_fbPlcCorrPoints[1].fX / 1000) + (GPx-x1)/dx * (_fbPlcCorrPoints[2].fX / 1000);
cx2 := (x2-GPx)/dx * (_fbPlcCorrPoints[3].fX / 1000) + (GPx-x1)/dx * (_fbPlcCorrPoints[4].fX / 1000);
cy1 := (x2-GPx)/dx * (_fbPlcCorrPoints[1].fY / 1000) + (GPx-x1)/dx * (_fbPlcCorrPoints[2].fY / 1000);
cy2 := (x2-GPx)/dx * (_fbPlcCorrPoints[3].fY / 1000) + (GPx-x1)/dx * (_fbPlcCorrPoints[4].fY / 1000);

// Interpolation in y
y1 := _fbPlcCorrPoints[1].fY_Ref / 1000;    // [mm -> m]
y2 := _fbPlcCorrPoints[3].fY_Ref / 1000;    // [mm -> m]
dy := y2-y1;
IF dy = 0 THEN (*F_Report_Error(ErrType:=EN_REPORT_ERROR_TYPE.Report_Error_0Pointer);*) RETURN; END_IF

// Calc interpolated 
CVx := (y2 - GPy)/dy * cx1 + (GPy-y1)/dy * cx2;
CVy := (y2 - GPy)/dy * cy1 + (GPy-y1)/dy * cy2;

// return accurate new correction only
dx_corr := CVx;
dy_corr := CVy;

calc_4p_correction := TRUE;
END_METHOD

(*
  Calculate grid point displacement for print unit banana deformation.
  2nd order approximation.
*)
METHOD PRIVATE calc_banana_correction : BOOL
VAR_INPUT
  x_pos   : LREAL;    // point x position [m]
  y_pos   : LREAL;    // point y position [m]
  fT1     : LREAL;    // temperature 1 [°C]
  fT2     : LREAL;    // temperature 2 [°C]
END_VAR
VAR_OUTPUT
  dx_corr : LREAL;    // point correction x [m]
END_VAR
VAR
  delta_T : LREAL;   // delta temperature
  e_max   : LREAL;   //
  a : LREAL;
  x_dash, y_dash : LREAL;
END_VAR
IF _y_max = 0 THEN RETURN; END_IF

x_dash := y_pos * 1000; // [m] -> [mm]

delta_T := fT2-fT1;
e_max   := delta_T * _e_max_per_deltaT;

a := 4 * e_max /  EXPT(_y_max, 2);
y_dash := a * EXPT(x_dash - (_y_max / 2), 2) - e_max;

// correction value
dx_corr := (y_dash / 1000);  // [mm] -> [m]

calc_banana_correction := TRUE;
END_METHOD

(*
  Calculate grid point displacement for a distortion with 4 rectangular defined points.
  Uses 2-bilinear interpolation between the 4 rectancular reference points.
*)
METHOD PRIVATE calc_PUC_4p_correction : BOOL
VAR_INPUT
  x_pos   : LREAL;    // point x position [m]
  y_pos   : LREAL;    // point y position [m]
END_VAR
VAR_OUTPUT
  dx_corr : LREAL;    // point correction x [m]
  dy_corr : LREAL;    // point correction y [m]
END_VAR
VAR
  dx, dy : LREAL;     // difference between Calibration Points (rectangle)
  x1, x2, y1, y2 : LREAL;
  cx1, cx2, cy1, cy2 : LREAL;
  GPx, GPy : LREAL;
  CVx, CVy : LREAL;
  lErrCtr : UDINT;
  
  pPUC_CorrPointsInd : POINTER TO ARRAY[1..4] OF ST_CORRECTION_POINT;
END_VAR
VAR CONSTANT
  fTranslateX : REAL := 1;
  fTranslateY : REAL := -1;
END_VAR
pPUC_CorrPointsInd := _pAdsCam^.pCorrectionPointsIndication;      // get points array from ADS
IF pPUC_CorrPointsInd = 0 THEN F_Report_Error(ErrType:=EN_REPORT_ERROR_TYPE.Report_Error_0Pointer);  RETURN; END_IF

// NOTE: the anchor points (poyx,posy) of the PUC points are set in WorkerCamera.mJobStart!

// Grid point position
GPx := x_pos; 
GPy := y_pos;

// Interpolation in x
x1 := pPUC_CorrPointsInd^[1].posx / 1000;    // [mm -> m]
x2 := pPUC_CorrPointsInd^[2].posx / 1000;    // [mm -> m]
dx := x2-x1;
IF dx = 0 THEN (*F_Report_Error(ErrType:=EN_REPORT_ERROR_TYPE.Report_Error_0Pointer);*) RETURN; END_IF

cx1 := (x2-GPx)/dx * ((pPUC_CorrPointsInd^[1].x * fTranslateX) / 1000) + (GPx-x1)/dx * ((pPUC_CorrPointsInd^[2].x * fTranslateX) / 1000);
cx2 := (x2-GPx)/dx * ((pPUC_CorrPointsInd^[3].x * fTranslateX) / 1000) + (GPx-x1)/dx * ((pPUC_CorrPointsInd^[4].x * fTranslateX) / 1000);
cy1 := (x2-GPx)/dx * ((pPUC_CorrPointsInd^[1].y * fTranslateY) / 1000) + (GPx-x1)/dx * ((pPUC_CorrPointsInd^[2].y * fTranslateY) / 1000);
cy2 := (x2-GPx)/dx * ((pPUC_CorrPointsInd^[3].y * fTranslateY) / 1000) + (GPx-x1)/dx * ((pPUC_CorrPointsInd^[4].y * fTranslateY) / 1000);

// Interpolation in y
y1 := pPUC_CorrPointsInd^[1].posy / 1000;    // [mm -> m]
y2 := pPUC_CorrPointsInd^[3].posy / 1000;    // [mm -> m]
dy := y2-y1;
IF dy = 0 THEN (*F_Report_Error(ErrType:=EN_REPORT_ERROR_TYPE.Report_Error_0Pointer);*) RETURN; END_IF

// Calc interpolated 
CVx := (y2 - GPy)/dy * cx1 + (GPy-y1)/dy * cx2;
CVy := (y2 - GPy)/dy * cy1 + (GPy-y1)/dy * cy2;

// return accurate new correction only
dx_corr := CVx;
dy_corr := CVy;

calc_PUC_4p_correction := TRUE;
END_METHOD

PROPERTY fT_PL1 : LREAL
SET
_fT1 := fT_PL1;
END_SET
END_PROPERTY

PROPERTY fT_PL2 : LREAL
SET
_fT2 := fT_PL2;
END_SET
END_PROPERTY

METHOD init : BOOL
VAR_INPUT
  pAdsCam        : POINTER TO FB_ADS_CAMERA;  // camera interface PUC
  fPxReso        : LREAL;   // pixel resolution
  fPuWidth       : LREAL;   // Print unit width [m]
END_VAR
_fPxResolution := fPxReso;
_y_max         := fPuWidth * 1000;  // -> [mm]
_pAdsCam       := pAdsCam;
IF _pAdsCam = 0 THEN LogError('missing _pAdsCam, ads interface unknown, call worker specific init before'); END_IF

// PU Deformation
_fbPlcCorrPoints[1].init(aName:='P1', aUnit:='mm', fX_Min:=-5, fX_Max:=5, fY_Min:=-5, fY_Max:=5, fIncrStep:=0.05, 
                        bButnInvertX:=TRUE, bButnInvertY:=TRUE, bValInvertX:=TRUE, bValInvertY:=FALSE);
_fbPlcCorrPoints[2].init(aName:='P2', aUnit:='mm', fX_Min:=-5, fX_Max:=5, fY_Min:=-5, fY_Max:=5, fIncrStep:=0.05,
                        bButnInvertX:=TRUE, bButnInvertY:=TRUE, bValInvertX:=TRUE, bValInvertY:=FALSE);
_fbPlcCorrPoints[3].init(aName:='P3', aUnit:='mm', fX_Min:=-5, fX_Max:=5, fY_Min:=-5, fY_Max:=5, fIncrStep:=0.05,
                        bButnInvertX:=TRUE, bButnInvertY:=TRUE, bValInvertX:=TRUE, bValInvertY:=FALSE);
_fbPlcCorrPoints[4].init(aName:='P4', aUnit:='mm', fX_Min:=-5, fX_Max:=5, fY_Min:=-5, fY_Max:=5, fIncrStep:=0.05,
                        bButnInvertX:=TRUE, bButnInvertY:=TRUE, bValInvertX:=TRUE, bValInvertY:=FALSE);
END_METHOD

(*
  Apply fine-alignement corrections to DefGrid point
*)
METHOD updateCorrection : BOOL
VAR_INPUT
  pPoint : POINTER TO ST_DeformationPointAccurate;
END_VAR
VAR
  x_pos, dx_corr, dx_tmp : LREAL; // [m]
  y_pos, dy_corr, dy_tmp : LREAL; // [m]
END_VAR
// grid point position
x_pos := F_SubPixelToMeter(lPosSubPx:=FC_LREAL_TO_DINT(pPoint^.x_ref), fResSubPx:=_fPxResolution);  // [px -> m] 
y_pos := F_SubPixelToMeter(lPosSubPx:=FC_LREAL_TO_DINT(pPoint^.y_ref), fResSubPx:=_fPxResolution);  // [px -> m]
dx_corr := 0;
dy_corr := 0;

// calc - 4 point sheet deformation (PU and machine mechanical distortions)
IF _bEnable_4p THEN
  calc_4p_correction(x_pos:=x_pos, y_pos:=y_pos, dx_corr=>dx_tmp, dy_corr=>dy_tmp);
  dx_corr := dx_tmp + dx_corr;
  dy_corr := dy_tmp + dy_corr;
END_IF

IF _bEnablePuc_4p THEN  (*PUC 4P correction used*)
  calc_PUC_4p_correction(x_pos:=x_pos, y_pos:=y_pos, dx_corr=>dx_tmp, dy_corr=>dy_tmp);
  dx_corr := dx_tmp + dx_corr;
  dy_corr := dy_tmp + dy_corr;
END_IF

// calc - banana correction
IF _bEnable_banana THEN
  calc_banana_correction(x_pos:=x_pos, y_pos:=y_pos, fT1:=_fT1, fT2:=_fT2, dx_corr=>dx_tmp);
  dx_corr := dx_tmp + dx_corr;
END_IF
// apply new correction to deformation correction 
pPoint^.dx := pPoint^.dx + F_MeterToSubPixelReal(fPosMeter:=dx_corr, fResoSubPx:=_fPxResolution);
pPoint^.dy := pPoint^.dy + F_MeterToSubPixelReal(fPosMeter:=dy_corr, fResoSubPx:=_fPxResolution);

updateCorrection := TRUE;
END_METHOD

END_FUNCTION_BLOCK

// ---- POUs/Print/DefGrid/FB_PointCorr.TcPOU
FUNCTION_BLOCK FB_PointCorr
VAR PERSISTENT
  _fX_Pos, _fX_Ref : LREAL;   // x position (correction / reference)
  _fY_Pos, _fY_Ref : LREAL;   // y position (correction / reference)
END_VAR
VAR
  bCmd_X_minus : BOOL;    // command x minus
  bCmd_X_plus  : BOOL;    // command x plus
  bCmd_Y_minus : BOOL;    // command y minus
  bCmd_Y_plus  : BOOL;    // command y plus
  bAny         : BOOL;    // any pressed
  tSlow, tFast : TON;
  rTrig        : R_TRIG;
  nIncr        : LREAL;
  nBtnColor    : UDINT;
  // settings (init)
  _aName       : STRING(3);   // name of element
  _aUnit       : STRING(10);  // element intended [unit]
  _fX_Min, _fX_Max : LREAL;   // limit x
  _fY_Min, _fY_Max : LREAL;   // limit y
  _fIncrStep    : LREAL;      // incr. step slow (stay on button), fast *10
  _bButnInvertX, _bButnInvertY : BOOL;  // change buttons
  _bValInvertX, _bValInvertY   : BOOL;  // value *-1
END_VAR
VAR CONSTANT
  RED          : UDINT := 16#FFFF0000;
  GREEN        : UDINT := 16#FF00FF00;
END_VAR

bAny := bCmd_X_minus OR bCmd_X_plus OR bCmd_Y_minus OR bCmd_Y_plus;
rTrig(CLK:=bAny);
tSlow(IN:=bAny AND NOT tSlow.Q, PT:=T#500MS);
tFast(IN:=bAny AND NOT rTrig.Q, PT:=T#2S);

IF    tFast.Q AND tSlow.Q THEN nIncr := 10*_fIncrStep;
ELSIF tSlow.Q OR rTrig.Q THEN nIncr := _fIncrStep;
ELSE               nIncr := 0;
END_IF

nBtnColor := GREEN;
//    button pressed     increment +/-                show limit
IF    (bCmd_X_minus AND NOT _bButnInvertX) OR (bCmd_X_plus  AND _bButnInvertX) THEN _fX_Pos := _fX_Pos - nIncr; IF _fX_Pos<=_fX_Min THEN nBtnColor:=RED; END_IF
ELSIF (bCmd_X_plus  AND NOT _bButnInvertX) OR (bCmd_X_minus AND _bButnInvertX) THEN _fX_Pos := _fX_Pos + nIncr; IF _fX_Pos>=_fX_Max THEN nBtnColor:=RED; END_IF
ELSIF (bCmd_Y_minus AND NOT _bButnInvertY) OR (bCmd_Y_plus  AND _bButnInvertY) THEN _fY_Pos := _fY_Pos - nIncr; IF _fY_Pos<=_fY_Min THEN nBtnColor:=RED; END_IF
ELSIF (bCmd_Y_plus  AND NOT _bButnInvertY) OR (bCmd_Y_minus AND _bButnInvertY) THEN _fY_Pos := _fY_Pos + nIncr; IF _fY_Pos>=_fY_Max THEN nBtnColor:=RED; END_IF
END_IF

// apply limit
IF _fX_Pos<=_fX_Min THEN _fX_Pos:=_fX_Min; END_IF
IF _fX_Pos>=_fX_Max THEN _fX_Pos:=_fX_Max; END_IF
IF _fY_Pos<=_fY_Min THEN _fY_Pos:=_fY_Min; END_IF
IF _fY_Pos>=_fY_Max THEN _fY_Pos:=_fY_Max; END_IF

(*correction value in X*)
PROPERTY fX : LREAL
GET
fX := SEL(_bValInvertX, _fX_Pos, -1*_fX_Pos);
END_GET
SET
_fX_Pos := SEL(_bValInvertX, fX, -1*fX);
END_SET
END_PROPERTY

PROPERTY fX_Ref : LREAL
GET
fX_Ref := _fX_Ref;
END_GET
SET
_fX_Ref := fX_Ref;
END_SET
END_PROPERTY

(*correction value in Y*)
PROPERTY fY : LREAL
GET
fY := SEL(_bValInvertY, _fY_Pos, -1*_fY_Pos);
END_GET
SET
_fY_Pos := SEL(_bValInvertY, fY, -1*fY);
END_SET
END_PROPERTY

PROPERTY fY_Ref : LREAL
GET
fY_Ref := _fY_Ref;
END_GET
SET
_fY_Ref := fY_Ref;
END_SET
END_PROPERTY

METHOD init : BOOL
VAR_INPUT
  aName : STRING(3);       // name
  aUnit : STRING(10);      // display unit
  fX_Min, fX_Max : LREAL;  // Limits
  fY_Min, fY_Max : LREAL;  // Limits
  fIncrStep      : LREAL;  // Increment step (slow) VISU
  bButnInvertX, bButnInvertY : BOOL;  // change buttons
  bValInvertX,  bValInvertY  : BOOL;  // value *-1
END_VAR
_aName := aName;
_aUnit := aUnit;
_fX_Min := fX_Min; _fX_Max := fX_Max;
_fY_Min := fY_Min; _fY_Max := fY_Max;
_fIncrStep := fIncrStep;
_bButnInvertX := bButnInvertX;
_bButnInvertY := bButnInvertY;
_bValInvertX := bValInvertX;
_bValInvertY := bValInvertY;
END_METHOD

END_FUNCTION_BLOCK

// ---- POUs/Print/DefGrid/FB_DefGridParamMediator.TcPOU
FUNCTION_BLOCK FB_DefGridParamMediator IMPLEMENTS I_ParamMediator
VAR
  _pCamWorker : POINTER TO FB_WorkerDefGrid_Camera;
  _pDefWorker : POINTER TO FB_WorkerDefGrid_Deformation;
  bInitOk     : BOOL;
END_VAR

METHOD init
VAR_INPUT
  pCamWorker : POINTER TO FB_WorkerDefGrid_Camera;
  pDefWorker : POINTER TO FB_WorkerDefGrid_Deformation;
END_VAR
IF pCamWorker <> 0 AND pCamWorker <> 0 THEN
  _pCamWorker := pCamWorker;
  _pDefWorker := pDefWorker;
  bInitOk := TRUE;
END_IF
END_METHOD

PROPERTY sCameraGridSettings : ST_CameraGridSettings
GET
IF bInitOk THEN
  sCameraGridSettings := _pCamWorker^.sCameraGridSettings;
END_IF
END_GET
END_PROPERTY

PROPERTY sDeformationGridSettings : ST_DefGridSettings
GET
IF bInitOk THEN
  sDeformationGridSettings := _pDefWorker^.sDeformationGridSettings;
END_IF
END_GET
END_PROPERTY

END_FUNCTION_BLOCK

// ---- POUs/Print/DefGrid/FB_WorkerDefGrid_Camera.TcPOU
FUNCTION_BLOCK FB_WorkerDefGrid_Camera EXTENDS FB_WorkerDefGrid IMPLEMENTS I_CameraSink
VAR
  // references
  _pAdsCam        : POINTER TO FB_ADS_CAMERA;
  _iParamMediator : I_ParamMediator;
  _fPrintUnitWidth : LREAL;
  
  // camera list
  _iCamList       : ARRAY[1..nMAXCAM] OF I_Camera; 
  _sCamName       : ARRAY[1..5] OF STRING;
  _nRegisteredCam : UDINT;    // number registered cameras
  _iActiveCam     : I_Camera; // active selected camera interface

  // cam status
  _bCamValid      : BOOL;
  _bCamReady      : BOOL;    // Camera no error
  _bConnectionOk  : BOOL;    //
  _bLineCamType   : BOOL;    // TRUE if it's a LineCamera
  _bSetInitCam    : BOOL;    // set initial camera
  _bCamStarted    : BOOL;    // Camera started
  
  // cam point status
  _bTeachOk       : BOOL;    // Teach successful
  _nTeachedPoints : UDINT;   // Teached points for this job
  _nScannedPoints : UDINT;   // Scanned points on current sheet
  _bCamDone       : BOOL;    //
  _nAddedPoint    : UDINT;   // point sent to image deformation on ct
  _nCamBufferPoints : UDINT;  // cam point input stream buffer (allows jittering the Attach of CT)
  _CamBufferPoints : ARRAY[1..GVL_Camera.cMaxNbMarks] OF ST_DeformationPointAccurate;
  
  // deformation status
  _eDeformationType            : E_DeformationType;
  _eDeformStep                 : E_DeformationStep;   // status deformation of ct
  _nCamDetected_X0             : DINT;                // detected sheet/repeat position [SubPx]  
  _fPrintLengthEffective       : LREAL;               // detected image length
  
  // Messages
  _pMsgConfig                  : POINTER TO ST_MSG_CONFIG;
  bCamNotAvailable             : BOOL;
  bCamModeNotSupported         : BOOL;
  fbMsg_CamNotAvailable        : FB_MESSAGE;
  fbMsg_CamModeNotSupported    : FB_MESSAGE;
  fbMsg_CamNoConnection        : FB_MESSAGE;
  
END_VAR

VAR PERSISTENT
  _fFeatureGrid   : LREAL := 2048;  // feature grid witdh (feature pich in x of cam frames), TODO: could be a normal var now
  _nActiveCam     : UDINT := 1;     // active camera selection
END_VAR

VAR CONSTANT
  nMAXCAM : UDINT := 5;
END_VAR

METHOD PRIVATE ActivateCamera : BOOL
VAR_INPUT
  iCam : I_Camera;
END_VAR
VAR
  i : UDINT;
END_VAR
IF iCam = 0 THEN F_Report_Error(ErrType:=EN_REPORT_ERROR_TYPE.Report_Error_0Pointer); RETURN; END_IF

IF _iActiveCam <> 0 THEN // Remove existing links
  _iActiveCam.DeactivateCam(iSink := THIS^);
END_IF

IF iCam.ActivateCam(iCameraSink := THIS^) THEN
  // get and set array index of registered cameras 
  FOR i :=1 TO _nRegisteredCam DO
    IF iCam = _iCamList[i] THEN
      _nActiveCam := i;              // set array index for visu/drop down
      EXIT; // select first found cam
    END_IF
  END_FOR
  _iActiveCam := iCam;        // set new cam
  ActivateCamera:=TRUE;
ELSE
  ActivateCamera:=FALSE;
END_IF
END_METHOD

METHOD AddCamPoint : BOOL
VAR_INPUT
	sDeformationPoint	: ST_DeformationPointAccurate;
END_VAR
IF _nCamBufferPoints >= GVL_Camera.cMaxNbMarks THEN LogError('AddCamPoint: CamPoint buffer is full (overflow), ignore point'); RETURN; END_IF

// add to internal buffer
_nCamBufferPoints := _nCamBufferPoints + 1;
_CamBufferPoints[_nCamBufferPoints] := sDeformationPoint; 

AddCamPoint := TRUE;
END_METHOD

METHOD AddTeachPoint : BOOL
VAR_INPUT
	sTeachPoint	: ST_DeformationPointAccurate;
END_VAR

// ignore the teach points for now

AddTeachPoint := TRUE;
END_METHOD

METHOD PROTECTED  Attach : BOOL
VAR_INPUT
  iCT              : I_CT;                         (*container at triggered event position*)
END_VAR
VAR
  bDeformErr : BOOL;
  eDeformStep : E_DeformationStep;
END_VAR
Attach := FALSE;
IF SUPER^.Attach(iCT:=iCT) THEN
  // OK, attached (enabled, was ok to be attached)
  IF _pNewAttached = 0 THEN RETURN; END_IF
  
  // Additional worker checks
  bDeformErr := _pNewAttached^.getDeformationStatus(eDStep=>eDeformStep);   // get latest status 
  // - deformation started? and no deformation error so far
  IF bDeformErr OR eDeformStep = E_DeformationStep.nothing THEN
    Release(iCT:=iCT);  // nothing to do anymore

  // - job is valid?
  ELSIF iCT.pJob = 0 OR NOT _bJobActive THEN
    _pNewAttached^.AbortDeformation(sReason:='No valid job', Src:=_pEcSrc^, bHideLog:=TRUE);
    Release(iCT:=iCT);

  // - camera ready
  ELSIF (NOT _bCamValid OR NOT _bCamReady) THEN  // check if cam is ready
    _pNewAttached^.AbortDeformation(sReason:='Camera invalid or not ready for attach', Src:=_pEcSrc^, bHideLog:=FALSE);
    Release(iCT:=iCT);

  // OK attach
  ELSE
    // start cam on ct
    LogLvl(Lvl:=E_LogSeverity.Debug, Msg:=F_Concat4('Start Camera with mode: ', TO_STRING(_iActiveCam.eCameraMode), ' on CT ', _pNewAttached^.print(0)));
    _pNewAttached^.StartCamera(eCameraMode:=_iActiveCam.eCameraMode, fFeatureGrid:=_fFeatureGrid, bResetDeformation:=TRUE);
  
    Attach := TRUE;
	END_IF
  
ELSE
  // parent attach failed case
END_IF
END_METHOD

PROPERTY bCamOk : BOOL
GET
bCamOk := _bCamValid;
END_GET
END_PROPERTY

PROPERTY bConnError : BOOL
GET
// TODO: propose the communication error on a better way.
bConnError := NOT _bConnectionOk;
END_GET
END_PROPERTY

PROPERTY bLineCamActive : BOOL
GET
bLineCamActive := _bLineCamType;
END_GET
END_PROPERTY

(*
  Event cam done "detecting points", sheet/repeate done.
  Called after last point will be streamed to same CT.
*)
METHOD CamDone : BOOL
IF _nAttachedCTs=0 OR NOT _bCamStarted OR _eDeformStep < E_DeformationStep.cameraStarted THEN
  // ignore done event if not started
  RETURN;
END_IF

// last point was received, we can dump the buffer and release the Container
streamPoints();   // stream all buffered points
IF _fPrintLengthEffective <> 0 THEN
  _pAttachedCt^.fPrintLengthEffective := _fPrintLengthEffective;
END_IF

LogLvl(Lvl:=E_LogSeverity.Debug, Msg:='CamDone');
Release(_pAttachedCt^);   // release head container

_bCamStarted := FALSE;
END_METHOD

(*
  Event cam started "detecting points".
  Is called before streaming cam points.
*)
METHOD CamStarted
VAR_INPUT
  nX0 : DINT; // detected start position
END_VAR
// erase rx buffer
_nCamBufferPoints := 0;
MEMSET(destAddr:=ADR(_CamBufferPoints[1]), fillByte:=0, n:=SIZEOF(_CamBufferPoints));

// save x0 for sheet lenght calculation
_nCamDetected_X0 := nX0;
_fPrintLengthEffective := 0;

_bCamStarted := TRUE;
END_METHOD

PROPERTY fCameraToPrintOffset : LREAL
GET
IF _iActiveCam <> 0 THEN
  fCameraToPrintOffset := _iActiveCam.fCameraToPrintOffset;
END_IF
END_GET
END_PROPERTY

PROPERTY fDetectToCamOffset : LREAL
GET
IF _iActiveCam <> 0 THEN
  fDetectToCamOffset := _iActiveCam.fDetectToCameraOffset;
END_IF
END_GET
END_PROPERTY

(* Detected "real" image lenght [m]*)
PROPERTY fPrintLengthEffective : LREAL
SET
_fPrintLengthEffective := fPrintLengthEffective;
END_SET
END_PROPERTY

METHOD Init
VAR_INPUT
  pMsgConfig : POINTER TO ST_MSG_CONFIG;         // message config
  fPrintResolution : LREAL := 1;                 // print(head) resolution in [dpi]
  fSubPxResolution : LREAL := 1;                 // SubPixel resolution [SubPx], resolution factor (fI_PrintResolution*fI_SubPxResolution=>Output resolution)
  bParallelCT : BOOL;                            // Support parallel processing of CTs
END_VAR
VAR
  lCtr : UDINT;
END_VAR
SUPER^.Init(pMsgConfig:=pMsgConfig, fPrintResolution:=fPrintResolution, fSubPxResolution:=fSubPxResolution, bParallelCT:=bParallelCT);

IF pMsgConfig = 0 THEN LogError('Init: invalid message config given'); END_IF 

(*Messaging*)
_pMsgConfig := pMsgConfig;

fbMsg_CamNotAvailable.pI_MsgConfig := _pMsgConfig;
fbMsg_CamNotAvailable.iI_MsgLocation := TO_INT(ePr_BLK_CAMERA);
fbMsg_CamNotAvailable.iI_MsgNumber := eC_STAG_CAM_NOTAVAIL;

fbMsg_CamModeNotSupported.pI_MsgConfig := _pMsgConfig;
fbMsg_CamModeNotSupported.iI_MsgLocation := TO_INT(ePr_BLK_CAMERA);
fbMsg_CamModeNotSupported.iI_MsgNumber := eC_STAG_CAM_MODE_NOTSUPPORTED; // camera not available

fbMsg_CamNoConnection.pI_MsgConfig := _pMsgConfig;
fbMsg_CamNoConnection.iI_MsgLocation := TO_INT(ePr_BLK_CAMERA);
fbMsg_CamNoConnection.iI_MsgNumber := eCMa_TCPIP_COMM_ERROR;    // tcpip connection error

_bConnectionOk := TRUE;
_bSetInitCam := TRUE; // request a default camera
END_METHOD

METHOD InitWorkerCamera
VAR_INPUT
  pAdsIf  : POINTER TO FB_ADS_CAMERA;
  iDefGridParamMediator : I_ParamMediator;
  fFeatureGrid : LREAL;   // feature grid with 
  fPrintUnitWidth   : LREAL;     // print unit width [m]
END_VAR
IF NOT bInitialized THEN LogError('Base Worker not initialized! call init() before'); RETURN; END_IF
IF pAdsIf = 0 THEN bInitialized := FALSE; LogError('Invalid parameter, no valid ads interface camera'); RETURN; END_IF
IF iDefGridParamMediator = 0 THEN bInitialized := FALSE; LogError('Invalid parameter, no valid param mediator'); RETURN; END_IF

_pAdsCam := pAdsIf;
_iParamMediator := iDefGridParamMediator;
_fPrintUnitWidth := fPrintUnitWidth;
_fFeatureGrid := fFeatureGrid;

_bCamStarted := FALSE;
// done by worker (always when cam activated)
//_bCamValid := _bCamReady := _bConnectionOk := FALSE;
//_nTeachedPoints := _nScannedPoints := 0;
END_METHOD

METHOD PRIVATE is_linecam : BOOL
VAR_INPUT
  sCamName : STRING;
END_VAR
is_linecam := SEL(FIND(F_ToLCase(sCamName), 'linecam') > 0, FALSE, TRUE);  // is it a LineCamera?
END_METHOD

METHOD   mJobStart
VAR_INPUT
	sJobDef	: CalmarCompPrint.I_JobDefinition;
END_VAR
VAR
  iNewCam : I_Camera;
  pCorrPointsInd : POINTER TO ARRAY[1..4] OF ST_CORRECTION_POINT;
END_VAR
IF _pAdsCam <> 0 THEN

  bCamNotAvailable := FALSE;
  bCamModeNotSupported := FALSE;

  // activate matching camera
  iNewCam := selectCamera(eNewCam:=_pAdsCam^.eCameraDevice);    // get camera settings from ADS
  IF NOT ActivateCamera(iCam:=iNewCam) THEN
    LogError(F_Concat2('Could not activate camera: ', TO_STRING(_pAdsCam^.eCameraDevice)));
    bCamNotAvailable := TRUE;
  ELSE
    // config camera from job
    _iActiveCam.fSubstrateLength := sJobDef.fImageDepth  / 1000;//sJobDef.fSubstrateDepth;      // [m]
    _iActiveCam.fSubstrateWidth  := sJobDef.fImageWidth  / 1000;//sJobDef.fSubstrateWidth;      // [m]
    _iActiveCam.fImageLength     := sJobDef.fImageDepth  / 1000;  // [mm] -> [m]
    _iActiveCam.fImageWidth      := sJobDef.fImageWidth  / 1000;  // [mm] -> [m]
    _iActiveCam.fFrameLength     := _fFeatureGrid;                // [px]
    bCamModeNotSupported := NOT _iActiveCam.setCameraMode(eCameraMode := _pAdsCam^.eCameraMode);     // set camera mode
    _iActiveCam.bEnableTrigger   := TRUE;    
    _iActiveCam.bManualTeach     := FALSE;
    _iActiveCam.mJobStart();

    // set deformation type based on camera
    _eDeformationType := selectDeformationType(_iActiveCam);
    
    // check settings
    IF _iActiveCam.fSubstrateLength = 0 THEN LogError('mJobStart() invalid SubstrateLength'); END_IF
    IF _iActiveCam.fSubstrateWidth = 0 THEN LogError('mJobStart() invalid SubstrateWidth'); END_IF
    IF _iActiveCam.fImageLength = 0 THEN LogError('mJobStart() invalid ImageLength'); END_IF
    IF _iActiveCam.fImageWidth = 0 THEN LogError('mJobStart() invalid ImageWidth'); END_IF
    
    // special case
    _bLineCamType := is_linecam(_iActiveCam.sName);  // is it a LineCamera?
  END_IF
  
  // set correction ref points (not done by PUC)
  pCorrPointsInd := _pAdsCam^.pCorrectionPointsIndication;
  IF pCorrPointsInd <> 0  THEN
    pCorrPointsInd^[1].posx := 0;
    pCorrPointsInd^[1].posy := LREAL_TO_REAL(((_fPrintUnitWidth * 1000) - sJobDef.fImageWidth) / 2);
    pCorrPointsInd^[2].posx := LREAL_TO_REAL(sJobDef.fImageDepth);
    pCorrPointsInd^[2].posy := LREAL_TO_REAL(((_fPrintUnitWidth * 1000) - sJobDef.fImageWidth) / 2);
    pCorrPointsInd^[3].posx := 0;
    pCorrPointsInd^[3].posy := LREAL_TO_REAL((((_fPrintUnitWidth * 1000) - sJobDef.fImageWidth) / 2) + sJobDef.fImageWidth);
    pCorrPointsInd^[4].posx := LREAL_TO_REAL(sJobDef.fImageDepth);
    pCorrPointsInd^[4].posy := LREAL_TO_REAL((((_fPrintUnitWidth * 1000) - sJobDef.fImageWidth) / 2) + sJobDef.fImageWidth);
  END_IF
END_IF

_bJobActive := TRUE;
END_METHOD

METHOD  mJobStop
VAR_INPUT
	sStatus	: CalmarCompPrint.I_JobStatus;
END_VAR
_bJobActive := FALSE;
END_METHOD

METHOD RegisterCamera : BOOL
VAR_INPUT
  iNewCam : I_Camera;
END_VAR
IF _nRegisteredCam < nMAXCAM AND iNewCam <> 0 THEN
  // configure message interface
  iNewCam.setMsgInterface(pMsgConfig:=_pMsgConfig);     // set message interface
  // add to internal list
  _nRegisteredCam := _nRegisteredCam + 1;
  _iCamList[_nRegisteredCam] := iNewCam;
  _sCamName[_nRegisteredCam] := iNewCam.sName;
  RegisterCamera := TRUE;
END_IF
END_METHOD

METHOD PRIVATE reviewState : BOOL
VAR
  bModeLowerThanRequested       : BOOL;
END_VAR
// review all camera states and set messages accordingly
IF _bJobActive AND _iActiveCam <> 0 THEN

  // -> mode less than desired
  IF _pAdsCam^.eCameraMode < _iActiveCam.eCameraMode THEN
    bModeLowerThanRequested := TRUE;
  END_IF

ELSE
  ;
END_IF
END_METHOD

PROPERTY sCameraGridSettings : ST_CameraGridSettings
GET
sCameraGridSettings.bValid := _bCamValid;
IF _bCamValid THEN
  sCameraGridSettings.eCameraMode := SEL(_iActiveCam<>0, E_CameraMode.NoCorrection, _iActiveCam.eCameraMode);
  sCameraGridSettings.eDeformationType := _eDeformationType;
  sCameraGridSettings.fGridFeaturePitch := _fFeatureGrid;
  sCameraGridSettings.fDetectToCam := SEL(_iActiveCam<>0,0,_iActiveCam.fDetectToCameraOffset);
END_IF
END_GET
END_PROPERTY

(*
  Select a registered camera from the requested device type.
*)
METHOD PRIVATE selectCamera : I_Camera
VAR_INPUT
  eNewCam  : E_CameraDevice;      // requested camera type
END_VAR
VAR
  bFound : BOOL;
  i : UDINT;
END_VAR
// select related camera (choose first matching)
bFound := FALSE;
FOR i :=1 TO _nRegisteredCam DO
  IF eNewCam = _iCamList[i].eDeviceType THEN
    // found
    selectCamera  := _iCamList[i]; // select new cam
    bFound := TRUE;
    EXIT; // select first found cam
	END_IF
END_FOR

IF NOT bFound THEN
  IF _iActiveCam <> 0 THEN
    // keep old if new was not found 
    LogError(F_Concat4('Try to select unavailable cam=', TO_STRING(eNewCam), ', use old cam=', TO_STRING(_iActiveCam.eDeviceType)));
  ELSIF _pAdsCam <> 0 THEN
    IF _iCamList[1] <> 0 THEN
      _iActiveCam := _iCamList[1];
      LogError(F_Concat4('Try to select unavailable cam=', TO_STRING(eNewCam), ', use other cam=', TO_STRING(_iActiveCam.eDeviceType)));
    ELSE
      LogError(F_Concat4('Try to select unavailable cam=', TO_STRING(eNewCam), ', no camera registered',''));
		END_IF
  END_IF
  
  selectCamera  := _iActiveCam; // return fallback camera 
END_IF
END_METHOD

(*
  Select deformation type (mode) based on selected camera device and camera mode.
*)
METHOD selectDeformationType : E_DeformationType
VAR_INPUT
  iCam : I_Camera;
END_VAR
IF    ( iCam.eCameraMode = E_CameraMode.Auto OR 
        iCam.eCameraMode = E_CameraMode.Live OR 
        iCam.eCameraMode = E_CameraMode.Trend
      ) AND ( 
        iCam.eDeviceType = E_CameraDevice.PrintMark
      )
THEN
  // local plc generated deformation, based on print marks
  selectDeformationType := E_DeformationType.LocalMarks1D;
  
ELSIF ( iCam.eCameraMode = E_CameraMode.Auto OR 
        iCam.eCameraMode = E_CameraMode.Live OR 
        iCam.eCameraMode = E_CameraMode.Trend 
      ) AND (
        iCam.eDeviceType = E_CameraDevice.Scanner OR 
        iCam.eDeviceType = E_CameraDevice.ScannerWithoutBackground
      ) 
THEN
  // live deformation done by py script
  IF iCam.eCameraMode = E_CameraMode.Trend THEN
    selectDeformationType := E_DeformationType.ScriptGridTrend;
  ELSE
    selectDeformationType := E_DeformationType.ScriptGrid;
	END_IF
  
ELSE
  // default no deformation
  selectDeformationType := E_DeformationType.NoDeformation;
END_IF
END_METHOD

METHOD setManualTeach
VAR_INPUT
  eCameraDevice    : E_CameraDevice;  
  fSubstrateLength : LREAL;   // teach substrate length
  fSubstrateWidth  : LREAL;   // teach substrate width
END_VAR
VAR
  iNewCam : I_Camera;
END_VAR
// activate Camera

iNewCam := selectCamera(eNewCam:=eCameraDevice);    // Scanner
IF NOT ActivateCamera(iCam:=iNewCam) THEN
  LogError(F_Concat2('Could not activate camera: ', TO_STRING(eCameraDevice)));
ELSE
  // config camera from manual teach
  _iActiveCam.fSubstrateLength := fSubstrateLength;
  _iActiveCam.fSubstrateWidth  := fSubstrateWidth;
  _iActiveCam.fImageLength     := fSubstrateLength;
  _iActiveCam.fImageWidth      := fSubstrateWidth;
  _iActiveCam.setCameraMode(eCameraMode :=E_CameraMode.Auto);     // set camera mode
  _iActiveCam.bEnableTrigger   := TRUE;   // enables trigger in CameraTrigger
  _iActiveCam.bManualTeach     := TRUE;   // enables manual trigger mode in CameraTrigger
  
  // special case
  _bLineCamType := is_linecam(_iActiveCam.sName);  // is it a LineCamera?
END_IF
END_METHOD

METHOD setupPosition
IF _pAttachedCt <> 0 THEN RETURN; END_IF    // Update only without attached container

fPosition := fDetectToCamOffset;
END_METHOD

METHOD PRIVATE streamPoints
VAR
  i : UDINT;
END_VAR
IF _nAttachedCTs=0 OR NOT _bCamStarted OR _eDeformStep < E_DeformationStep.cameraStarted THEN
  RETURN;
END_IF


// stream buffered points
_nAddedPoint := _pAttachedCt^.nRegisteredCameraPoints;

WHILE _nAddedPoint < _nCamBufferPoints DO
  
  // apply detected X0 position
  IF _nAddedPoint = 0 THEN 
    IF _pAttachedCt^.nPosPrint_X0 <> _nCamDetected_X0 THEN
      LogWarning(F_Concat5('streamPoints: CamDetected X0=', TO_STRING(_nCamDetected_X0), '<>CT X0', TO_STRING(_pAttachedCt^.nPosPrint_X0), '!'));
    END_IF
	END_IF
  // apply cam point to CT
  IF _pAttachedCt^.AddCamPoint(sPoint:=_CamBufferPoints[_nAddedPoint+1]) THEN 
    //cameraImgProc(newDeformationPoint:=iDeformationPoint);  //Update image processing
  ELSE
    LogError(Msg:='addCamPoint failed, add to CT error');
  END_IF;
  
  // added
  _nAddedPoint :=_nAddedPoint+1;
END_WHILE
END_METHOD

METHOD  work
IF _iParamMediator = 0 THEN RETURN; END_IF

SUPER^.work();


//-----------------------------------------------------------
//- automatic worker setup & control
IF _bSetInitCam AND _iActiveCam = 0 THEN    // try to set a default camera at start
  ActivateCamera(selectCamera(eNewCam:=E_CameraDevice.SheetDetect));
  _bSetInitCam := FALSE;
  _bCamValid := TRUE;

ELSIF _iActiveCam <> 0 THEN                 // a camera is activated
  
  // --- cyclic call always when cam is active ---
  _bCamValid := TRUE;
  
  //-- update status
  _bCamReady := _iActiveCam.GetCamStatus(
                              bConnectionOK  => _bConnectionOk, 
                              bTeachOk       => _bTeachOk, 
                              nTeachedPoints => _nTeachedPoints, 
                              nScannedPoints => _nScannedPoints,
                              //bCamStarted  => _bCamStarted,   // we use done event from I_CameraSink (TODO: review with LineCam!)
                              bCamDone       => _bCamDone
                            );
  // -- worker position setup
  setupPosition();
ELSE
  _bCamValid := FALSE;                    // invalid camera
END_IF


// -----------------------------------------------------------
// Work only with attached container
IF _pAttachedCt <> 0 THEN

  // we have a HEAD container
  bError := _pAttachedCt^.getDeformationStatus(eDStep => _eDeformStep);
  
    IF _eDeformStep > E_DeformationStep.nothing AND _bCamReady AND _bTeachOk THEN      // start only if previous started
      (*done during attach: 
      IF _eDeformStep < E_DeformationStep.cameraStarted THEN
        // start cam on ct
        LogLvl(Lvl:=E_LogSeverity.Debug, Msg:=F_Concat2('Start Camera with mode: ', TO_STRING(_iActiveCam.eCameraMode)));
        _pAttachedCt^.StartCamera(eCameraMode:=_iActiveCam.eCameraMode, fFeatureGrid:=_fFeatureGrid);
      *)
			IF _eDeformStep >= E_DeformationStep.cameraStarted AND _bCamStarted THEN
        // run update on ct
        // stream points
        streamPoints();
        // superview abort cases
      END_IF
      
      // NOTE: Release() is done in CamDone() method
    ELSE
      IF _bCamStarted THEN
        // error on camera while started
        LogError('Abort Camera while it was started');
			END_IF
      // release because cam not ready or pior worker not done its job
      Release(_pAttachedCt^);   // release head container
		END_IF

END_IF

// call messages
fbMsg_CamNotAvailable    (bI_Status:=bCamNotAvailable);
fbMsg_CamModeNotSupported(bI_Status:=bCamModeNotSupported);
fbMsg_CamNoConnection    (bI_Status:=NOT _bConnectionOk);
END_METHOD

END_FUNCTION_BLOCK

// ---- POUs/Print/DefGrid/FB_WorkerDefGrid.TcPOU
FUNCTION_BLOCK ABSTRACT FB_WorkerDefGrid EXTENDS FB_Worker
VAR_OUTPUT
  bError            : BOOL;                           // an error is active
  nError            : UDINT;                          // error code if error active, =0 else
END_VAR
VAR
  // config
  _pMsgConfigExt    : POINTER TO ST_MSG_CONFIG;       // external message config (puc message interface)
  _fPrintResolution : LREAL := 1;                     // print(head) resolution in [dpi]
  _fSubPxResolution : LREAL := 1;                     // SubPixel resolution [SubPx], resolution factor (fI_PrintResolution*fI_SubPxResolution=>Output resolution
  _name             : STRING;                         // Worker name
  _sVisuName        : STRING := 'VISU_WorkerDefGrid'; // Worker visu instance name
  _pEcSrc           : POINTER TO T_ErrSrc;            // Error source definition

  // job
  _bJobActive       : BOOL;                           // a job is active
  // ct
  _bAttached        : BOOL;                           // one ct is attached
  _pAttachedCt      : POINTER TO FB_ContainerDefGrid; // currently attached container (HEAD)
  _pNewAttached     : POINTER TO FB_ContainerDefGrid; // last attached container (as return value of Attach() (TAIL))
  _pNewAttachedHdlData : POINTER TO ST_WorkerDefGrid_CTData;  // pointer to handling data for last attached
  _bSupportParallelCT : BOOL := FALSE;                // support for parallel CTs (else avoid attach while one connected).
  _nAttachedCTs     : UDINT;                          // Number of currently attached CTs
  _nHeadCtId        : DINT;                           // ID of CT at Attached Head
  _pAttachedCTList  : ARRAY[nLowerIndexCTList..nUpperIndexCTList] OF POINTER TO FB_ContainerDefGrid;    // current attached CTs
  _stAttachedCTData : ARRAY[nLowerIndexCTList..nUpperIndexCTList] OF ST_WorkerDefGrid_CTData;           // additional "handling" data per attached CT
  // position control
  fCtPosition       : LREAL;     // Container position relative to worker position
  _bForceRelease    : BOOL;                           // Manually force a ct release

  // view
  nGridRowStart, nGridColStart: UDINT := 0;
END_VAR
VAR_STAT
  // static variables, SAME for ALL Workers
  _pCTM             : POINTER TO FB_CTManagerDefGrid;             // "Global" Container Manager
  _fCtSecurityReleasePos : LREAL := 0;                // [SubPx] position where to release current ct at last (security release)
END_VAR
VAR PERSISTENT
  _fWorkerPosition  : LREAL;                          // [m] worker distance to X0 (position from X0) (CT creation X0 and domain)
END_VAR
VAR CONSTANT
  // list size
  nLowerIndexCTList : UDINT := 1;
  nUpperIndexCTList : UDINT := 4; 
END_VAR

(*
  Generic abort implementation of DefGrid CT.
*)
METHOD Abort
VAR_INPUT
  iCT       : I_CT;
  sReason   : STRING;
END_VAR
VAR
  _pCt   : POINTER TO FB_ContainerDefGrid;
  eStep     : E_DeformationStep;
END_VAR
IF iCT = 0 AND _pAttachedCt <> 0 THEN             // no ct given and check if one is attached 
  _pCt := _pAttachedCt;
ELSIF getCtInst(iCT:=iCT, pCT=>_pCt) = 0 THEN     // get specific container from given interface
  RETURN; 
END_IF

IF _pCt = 0 THEN RETURN; END_IF
  
// abort CT
  // Do generic known aborts on CT
  // - Deformation
  _pCt^.getDeformationStatus(eDStep=>eStep);
  IF eStep >= E_DeformationStep.nothing THEN
    _pCt^.AbortDeformation(sReason:=sReason, Src:=_pEcSrc^, bHideLog:=FALSE);
  
END_IF
END_METHOD

METHOD PROTECTED  Attach : BOOL
VAR_INPUT
  iCT       : I_CT;            (*container at triggered event position*)
END_VAR
VAR
  i : UDINT;
END_VAR
Attach := FALSE;

IF iCT = 0 THEN
  LogError(Msg:='attach failed -> not ct given');
  
ELSIF bWorkerEnable THEN  // worker enabled
  
  IF getCtInst(iCT:=iCT, pCT=>_pNewAttached) <> 0 THEN    // get specific container
    // add to list ()
    IF push(pNewCT:=_pNewAttached) THEN 
      LogLvl(Lvl:=E_LogSeverity.Debug, Msg:=F_Concat4('Attach CT[', TO_STRING(_nAttachedCTs), ']: ', _pNewAttached^.print(0)));
      Attach:=TRUE;                                 // attach new
    END_IF
  ELSE
    LogError(Msg:='attach failed: could not get CT instance');
  END_IF

ELSIF NOT bWorkerEnable AND _nAttachedCTs > 0 THEN // disabled and already a CT attached
  // force release all attached CT, and ignore attach
  LogLvl(Lvl:=E_LogSeverity.Debug, Msg:='Worker disabled flush list of all attached CT');
  WHILE _nAttachedCTs > 0 DO
    Release(iCT:=_pAttachedCt^);
	END_WHILE

ELSIF NOT bWorkerEnable AND _pAttachedCt = 0 THEN  
  ;   // nothing to do, ignore attach

ELSE      // unspecified (error)case just log it
  LogError(Msg:='not tracked case');
END_IF


// ok to attach
END_METHOD

{attribute 'monitoring':='call'}
PROPERTY bAttached : BOOL
GET
bAttached := _bAttached;
END_GET
END_PROPERTY

{attribute 'monitoring':='call'}
PROPERTY fPosition : LREAL
GET
fPosition := _fWorkerPosition;
END_GET
SET
_fWorkerPosition := fPosition;  // [m] save position
END_SET
END_PROPERTY

(*
  Get specific container from interface.
  Returns specific container in return value and output parameter.
*)
METHOD INTERNAL getCtInst : POINTER TO FB_ContainerDefGrid
VAR_INPUT
  iCT              : I_CT;                         (*container at triggered event position*)
END_VAR
VAR_OUTPUT
  pCT              : POINTER TO FB_ContainerDefGrid;
END_VAR
IF NOT bInitialized THEN RETURN; END_IF
IF _pCTM = 0 THEN RETURN; END_IF

pCT := 0;
getCtInst := _pCTM^.GetContainerInstance(iCT);   // get real ct fb inst
IF getCtInst <> 0 THEN
  pCT := getCtInst;   // OK all good
ELSE
  LogError(Msg:='specific container not found');
END_IF
END_METHOD

(*
  Get relative position to this worker (relative to track position)
*)
METHOD getPosRelToAttach : DINT
VAR_INPUT
  iCT : I_CT;
END_VAR
// relative position to X0 - tracking offset of this worker
getPosRelToAttach := iCT.GetPosRel(iTracker:=_iCTTracker) - _nTrackOffset;
END_METHOD

METHOD Init
VAR_INPUT
  pMsgConfig : POINTER TO ST_MSG_CONFIG;         // message config
  fPrintResolution : LREAL := 1;                 // print(head) resolution in [dpi]
  fSubPxResolution : LREAL := 1;                 // SubPixel resolution [SubPx], resolution factor (fI_PrintResolution*fI_SubPxResolution=>Output resolution)
  bParallelCT : BOOL;                            // Support parallel processing of CTs
END_VAR
VAR

END_VAR
_bAttached := 0;
_pAttachedCt := 0;
_nAttachedCTs := 0;

IF _pCTM = 0 THEN LogError(Msg:='Init: invalid parameter'); RETURN; END_IF

// save config
_pMsgConfigExt := pMsgConfig;
_fPrintResolution := fPrintResolution;
_fSubPxResolution := fSubPxResolution;
_fCtSecurityReleasePos := 0;
_bSupportParallelCT := bParallelCT;

setName('');

// init error source reference
_pEcSrc := ErrorCodes.fbErrCodeMngr.registerErrSource(
  nLocId := 0,
  aInstPath := InstanceName,
  aLocDescr := _name
);
IF _pEcSrc = 0 THEN LogError('could not register error source'); END_IF

bInitialized := TRUE;
END_METHOD

METHOD ABSTRACT mJobStart
VAR_INPUT
	sJobDef	: CalmarCompPrint.I_JobDefinition;
END_VAR
// implement in parent class
END_METHOD

METHOD ABSTRACT mJobStop
VAR_INPUT
	sStatus	: CalmarCompPrint.I_JobStatus;
END_VAR
END_METHOD

PROPERTY pCTM : POINTER TO FB_CTManagerDefGrid
GET
pCTM := _pCTM;
END_GET
SET
_pCTM := pCTM;
END_SET
END_PROPERTY

METHOD PRIVATE pull : BOOL
VAR_INPUT
  pRemCT : POINTER TO FB_ContainerDefGrid;
END_VAR
VAR_OUTPUT
  nRemIndex : DINT := 0;
END_VAR
VAR
  i                : DINT;
  Index            : DINT;
  LowerIndex       : DINT := 1;
END_VAR
IF _nAttachedCTs = 0 THEN LogError('Release: but no CT is attached'); RETURN; END_IF

// -- find if ct is in attached list
Index := -1;
FOR i:= TO_DINT(nLowerIndexCTList) TO TO_DINT(nLowerIndexCTList + _nAttachedCTs - 1) DO
  IF _pAttachedCTList[i] = pRemCT THEN
    Index := i;
    EXIT;     // found
  END_IF
END_FOR
IF Index = -1 THEN LogError('Release: ct inst not found in list'); RETURN; END_IF

// do stop CT callback if removing first
IF Index = TO_DINT(nLowerIndexCTList) THEN StopCT(pCtDefGrid:=pRemCT); END_IF

// compress list
IF Index >= TO_DINT(nLowerIndexCTList) AND Index < TO_DINT(nUpperIndexCTList) THEN
  // - ct references
  MEMMOVE(              // shift all above entries down
    destAddr := ADR( _pAttachedCTList[Index] ), 
    srcAddr  := ADR( _pAttachedCTList[Index + 1] ), 
    n        := DINT_TO_UDINT(SIZEOF(_pAttachedCTList[LowerIndex]) * (UDINT_TO_DINT(_nAttachedCTs) - Index - 1 + LowerIndex))
  );
  _pAttachedCTList[nUpperIndexCTList] := 0;     // erase last(compressed) list entry
  // - ct handling data
  MEMMOVE(              // shift all above entries down
    destAddr := ADR( _stAttachedCTData[Index] ), 
    srcAddr  := ADR( _stAttachedCTData[Index + 1] ), 
    n        := DINT_TO_UDINT(SIZEOF(_stAttachedCTData[LowerIndex]) * (UDINT_TO_DINT(_nAttachedCTs) - Index - 1 + LowerIndex))
  );
  MEMSET(destAddr:=ADR(_stAttachedCTData[nUpperIndexCTList]), fillByte:=0, n:=SIZEOF(_stAttachedCTData[1]));  // erase last(compressed) list entry
END_IF
_pAttachedCTList[_nAttachedCTs] := 0;   // erase last element
MEMSET(destAddr:=ADR(_stAttachedCTData[_nAttachedCTs]), fillByte:=0, n:=SIZEOF(_stAttachedCTData[1]));  // erase last element
  
// remove
_nAttachedCTs := _nAttachedCTs - 1;   // remove one element

IF _nAttachedCTs > 0 THEN 
  // Start new HEAD
  _pAttachedCt := _pAttachedCTList[1];
  _bAttached := TRUE;
  StartCT(pCtDefGrid:=_pAttachedCt);
ELSE
  // CT list empty (no ct attached)
  _pAttachedCt := 0;
  _bAttached := 0;
END_IF

nRemIndex := Index;
pull := TRUE;
END_METHOD

